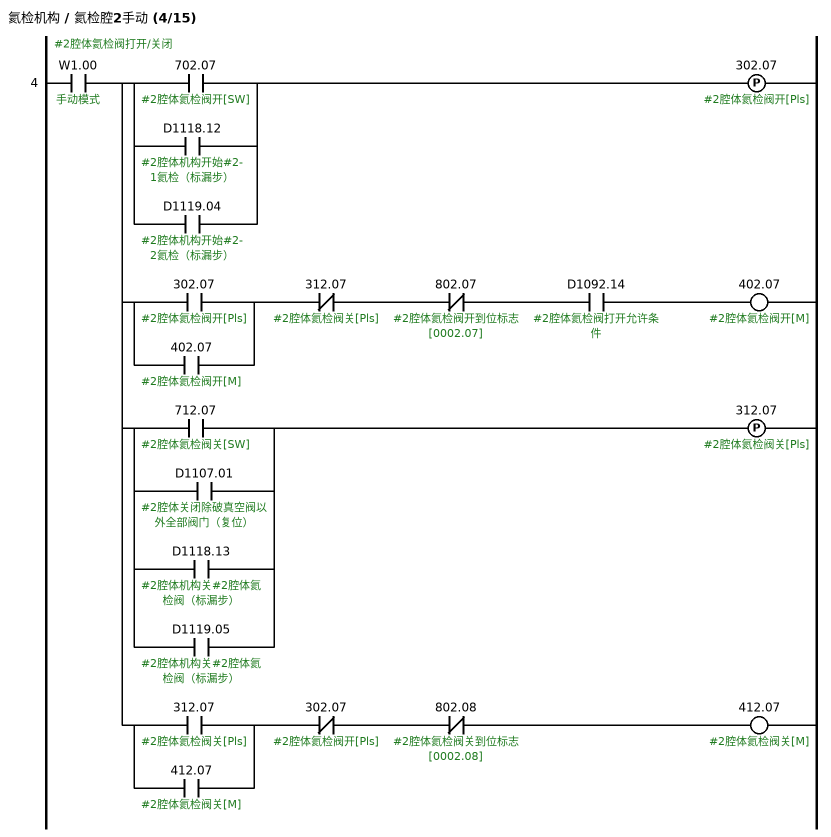
; [picture p168: 氦检机构 / 氦检腔2手动, rungs 4-4]
; rung 4: #2腔体氦检阀打开/关闭
LD W1.00  ; 手动模式
OUT TR0
LD 702.07  ; #2腔体氦检阀开[SW]
OR D1118.12  ; #2腔体机构开始#2-1氦检（标漏步）
OR D1119.04  ; #2腔体机构开始#2-2氦检（标漏步）
ANDLD
DIFU(013) 302.07  ; #2腔体氦检阀开[Pls]
LD TR0
LD 302.07  ; #2腔体氦检阀开[Pls]
OR 402.07  ; #2腔体氦检阀开[M]
ANDLD
ANDNOT 312.07  ; #2腔体氦检阀关[Pls]
ANDNOT 802.07  ; #2腔体氦检阀开到位标志[0002.07]
AND D1092.14  ; #2腔体氦检阀打开允许条件
OUT 402.07  ; #2腔体氦检阀开[M]
LD TR0
LD 712.07  ; #2腔体氦检阀关[SW]
OR D1107.01  ; #2腔体关闭除破真空阀以外全部阀门（复位）
OR D1118.13  ; #2腔体机构关#2腔体氦检阀（标漏步）
OR D1119.05  ; #2腔体机构关#2腔体氦检阀（标漏步）
ANDLD
DIFU(013) 312.07  ; #2腔体氦检阀关[Pls]
LD TR0
LD 312.07  ; #2腔体氦检阀关[Pls]
OR 412.07  ; #2腔体氦检阀关[M]
ANDLD
ANDNOT 302.07  ; #2腔体氦检阀开[Pls]
ANDNOT 802.08  ; #2腔体氦检阀关到位标志[0002.08]
OUT 412.07  ; #2腔体氦检阀关[M]

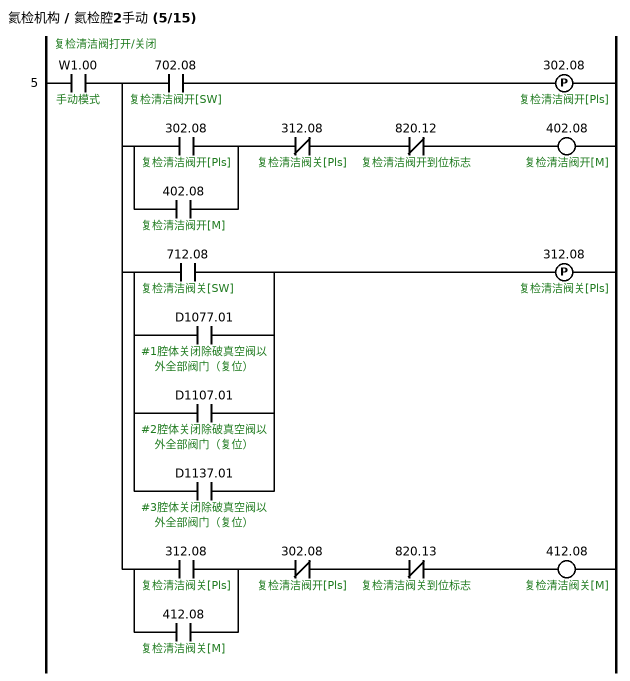
; rung 5: 复检清洁阀打开/关闭
LD W1.00  ; 手动模式
OUT TR0
AND 702.08  ; 复检清洁阀开[SW]
DIFU(013) 302.08  ; 复检清洁阀开[Pls]
LD TR0
LD 302.08  ; 复检清洁阀开[Pls]
OR 402.08  ; 复检清洁阀开[M]
ANDLD
ANDNOT 312.08  ; 复检清洁阀关[Pls]
ANDNOT 820.12  ; 复检清洁阀开到位标志
OUT 402.08  ; 复检清洁阀开[M]
LD TR0
LD 712.08  ; 复检清洁阀关[SW]
OR D1077.01  ; #1腔体关闭除破真空阀以外全部阀门（复位）
OR D1107.01  ; #2腔体关闭除破真空阀以外全部阀门（复位）
OR D1137.01  ; #3腔体关闭除破真空阀以外全部阀门（复位）
ANDLD
DIFU(013) 312.08  ; 复检清洁阀关[Pls]
LD TR0
LD 312.08  ; 复检清洁阀关[Pls]
OR 412.08  ; 复检清洁阀关[M]
ANDLD
ANDNOT 302.08  ; 复检清洁阀开[Pls]
ANDNOT 820.13  ; 复检清洁阀关到位标志
OUT 412.08  ; 复检清洁阀关[M]

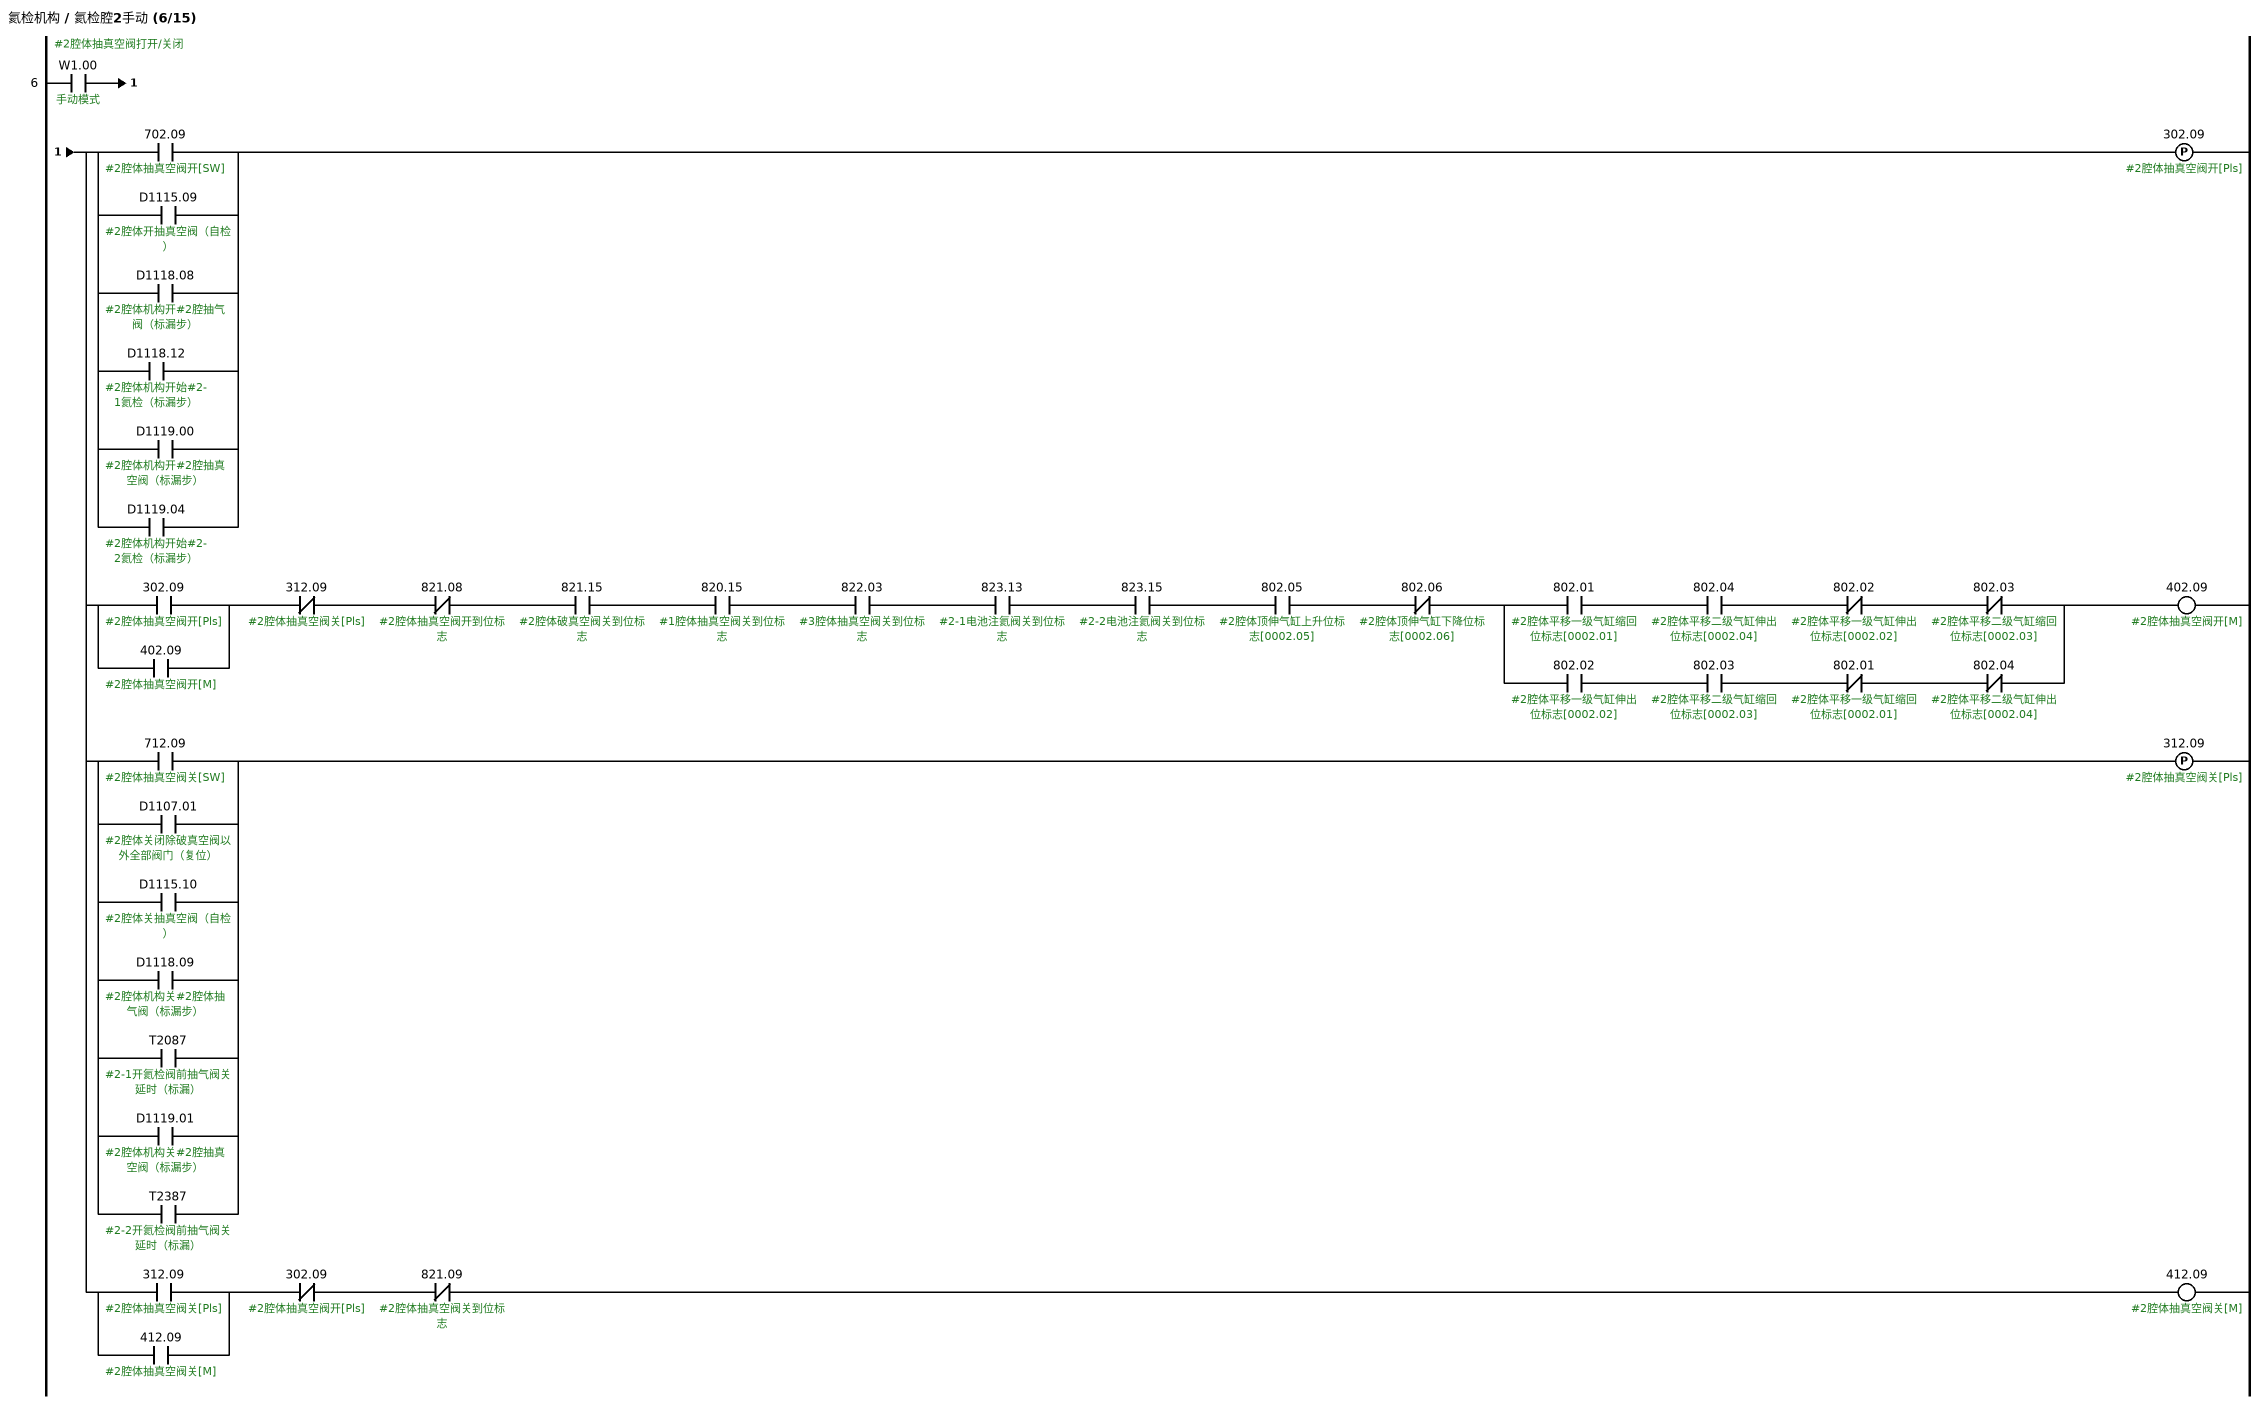
; rung 6: #2腔体抽真空阀打开/关闭
LD W1.00  ; 手动模式
OUT TR0
LD 702.09  ; #2腔体抽真空阀开[SW]
OR D1115.09  ; #2腔体开抽真空阀（自检）
OR D1118.08  ; #2腔体机构开#2腔抽气阀（标漏步）
OR D1118.12  ; #2腔体机构开始#2-1氦检（标漏步）
OR D1119.00  ; #2腔体机构开#2腔抽真空阀（标漏步）
OR D1119.04  ; #2腔体机构开始#2-2氦检（标漏步）
ANDLD
DIFU(013) 302.09  ; #2腔体抽真空阀开[Pls]
LD TR0
LD 302.09  ; #2腔体抽真空阀开[Pls]
OR 402.09  ; #2腔体抽真空阀开[M]
ANDLD
ANDNOT 312.09  ; #2腔体抽真空阀关[Pls]
ANDNOT 821.08  ; #2腔体抽真空阀开到位标志
AND 821.15  ; #2腔体破真空阀关到位标志
AND 820.15  ; #1腔体抽真空阀关到位标志
AND 822.03  ; #3腔体抽真空阀关到位标志
AND 823.13  ; #2-1电池注氦阀关到位标志
AND 823.15  ; #2-2电池注氦阀关到位标志
AND 802.05  ; #2腔体顶伸气缸上升位标志[0002.05]
ANDNOT 802.06  ; #2腔体顶伸气缸下降位标志[0002.06]
LD 802.01  ; #2腔体平移一级气缸缩回位标志[0002.01]
AND 802.04  ; #2腔体平移二级气缸伸出位标志[0002.04]
ANDNOT 802.02  ; #2腔体平移一级气缸伸出位标志[0002.02]
ANDNOT 802.03  ; #2腔体平移二级气缸缩回位标志[0002.03]
LD 802.02  ; #2腔体平移一级气缸伸出位标志[0002.02]
AND 802.03  ; #2腔体平移二级气缸缩回位标志[0002.03]
ANDNOT 802.01  ; #2腔体平移一级气缸缩回位标志[0002.01]
ANDNOT 802.04  ; #2腔体平移二级气缸伸出位标志[0002.04]
ORLD
ANDLD
OUT 402.09  ; #2腔体抽真空阀开[M]
LD TR0
LD 712.09  ; #2腔体抽真空阀关[SW]
OR D1107.01  ; #2腔体关闭除破真空阀以外全部阀门（复位）
OR D1115.10  ; #2腔体关抽真空阀（自检）
OR D1118.09  ; #2腔体机构关#2腔体抽气阀（标漏步）
OR T2087  ; #2-1开氦检阀前抽气阀关延时（标漏）
OR D1119.01  ; #2腔体机构关#2腔抽真空阀（标漏步）
OR T2387  ; #2-2开氦检阀前抽气阀关延时（标漏）
ANDLD
DIFU(013) 312.09  ; #2腔体抽真空阀关[Pls]
LD TR0
LD 312.09  ; #2腔体抽真空阀关[Pls]
OR 412.09  ; #2腔体抽真空阀关[M]
ANDLD
ANDNOT 302.09  ; #2腔体抽真空阀开[Pls]
ANDNOT 821.09  ; #2腔体抽真空阀关到位标志
OUT 412.09  ; #2腔体抽真空阀关[M]

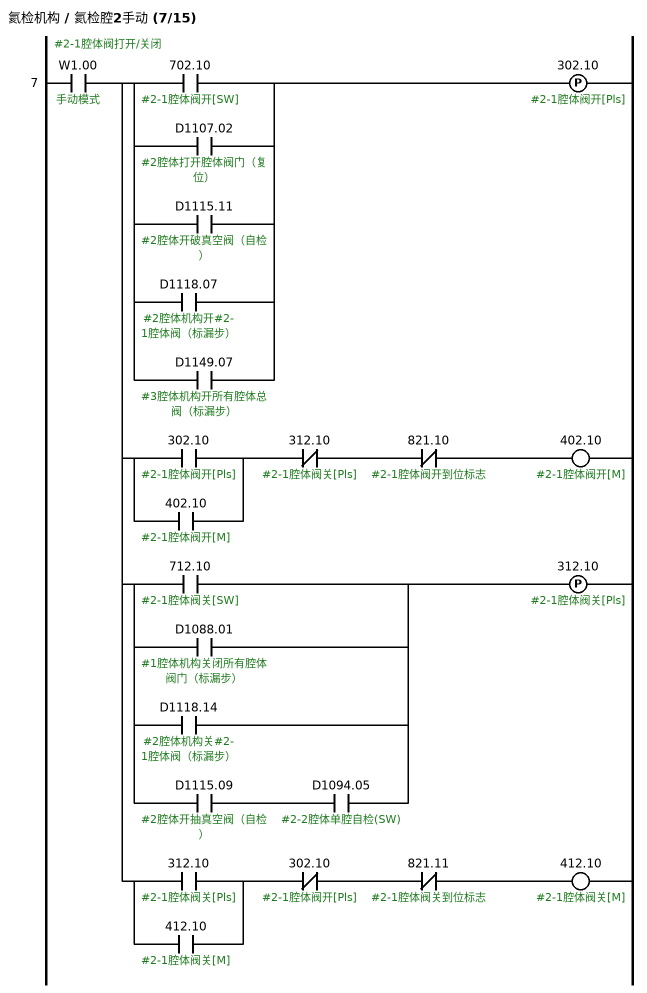
; rung 7: #2-1腔体阀打开/关闭
LD W1.00  ; 手动模式
OUT TR0
LD 702.10  ; #2-1腔体阀开[SW]
OR D1107.02  ; #2腔体打开腔体阀门（复位）
OR D1115.11  ; #2腔体开破真空阀（自检）
OR D1118.07  ; #2腔体机构开#2-1腔体阀（标漏步）
OR D1149.07  ; #3腔体机构开所有腔体总阀（标漏步）
ANDLD
DIFU(013) 302.10  ; #2-1腔体阀开[Pls]
LD TR0
LD 302.10  ; #2-1腔体阀开[Pls]
OR 402.10  ; #2-1腔体阀开[M]
ANDLD
ANDNOT 312.10  ; #2-1腔体阀关[Pls]
ANDNOT 821.10  ; #2-1腔体阀开到位标志
OUT 402.10  ; #2-1腔体阀开[M]
LD TR0
LD 712.10  ; #2-1腔体阀关[SW]
OR D1088.01  ; #1腔体机构关闭所有腔体阀门（标漏步）
OR D1118.14  ; #2腔体机构关#2-1腔体阀（标漏步）
LD D1115.09  ; #2腔体开抽真空阀（自检）
AND D1094.05  ; #2-2腔体单腔自检(SW)
ORLD
ANDLD
DIFU(013) 312.10  ; #2-1腔体阀关[Pls]
LD TR0
LD 312.10  ; #2-1腔体阀关[Pls]
OR 412.10  ; #2-1腔体阀关[M]
ANDLD
ANDNOT 302.10  ; #2-1腔体阀开[Pls]
ANDNOT 821.11  ; #2-1腔体阀关到位标志
OUT 412.10  ; #2-1腔体阀关[M]

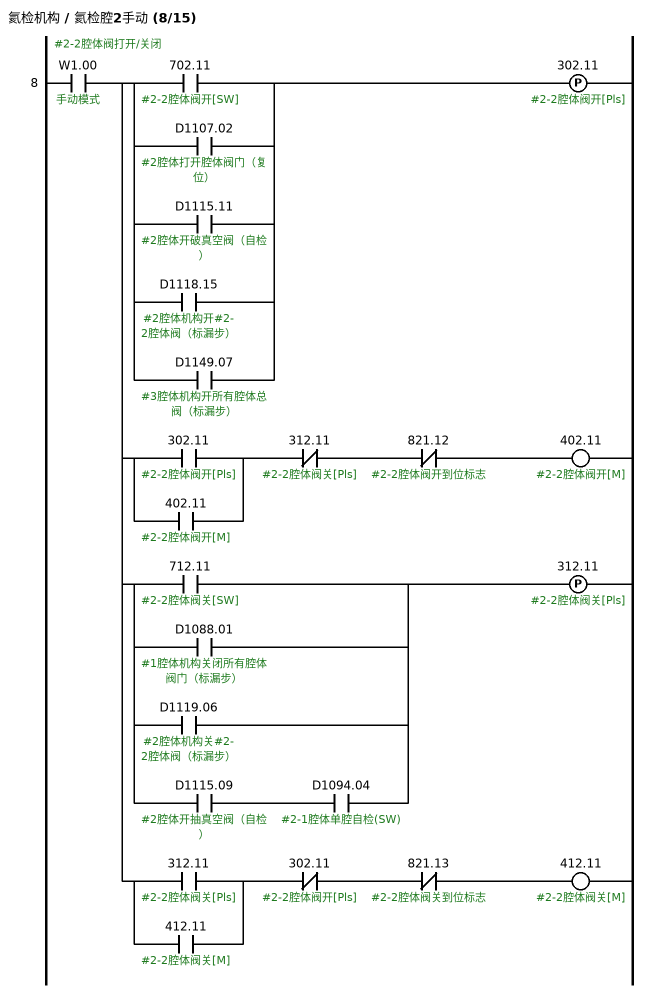
; rung 8: #2-2腔体阀打开/关闭
LD W1.00  ; 手动模式
OUT TR0
LD 702.11  ; #2-2腔体阀开[SW]
OR D1107.02  ; #2腔体打开腔体阀门（复位）
OR D1115.11  ; #2腔体开破真空阀（自检）
OR D1118.15  ; #2腔体机构开#2-2腔体阀（标漏步）
OR D1149.07  ; #3腔体机构开所有腔体总阀（标漏步）
ANDLD
DIFU(013) 302.11  ; #2-2腔体阀开[Pls]
LD TR0
LD 302.11  ; #2-2腔体阀开[Pls]
OR 402.11  ; #2-2腔体阀开[M]
ANDLD
ANDNOT 312.11  ; #2-2腔体阀关[Pls]
ANDNOT 821.12  ; #2-2腔体阀开到位标志
OUT 402.11  ; #2-2腔体阀开[M]
LD TR0
LD 712.11  ; #2-2腔体阀关[SW]
OR D1088.01  ; #1腔体机构关闭所有腔体阀门（标漏步）
OR D1119.06  ; #2腔体机构关#2-2腔体阀（标漏步）
LD D1115.09  ; #2腔体开抽真空阀（自检）
AND D1094.04  ; #2-1腔体单腔自检(SW)
ORLD
ANDLD
DIFU(013) 312.11  ; #2-2腔体阀关[Pls]
LD TR0
LD 312.11  ; #2-2腔体阀关[Pls]
OR 412.11  ; #2-2腔体阀关[M]
ANDLD
ANDNOT 302.11  ; #2-2腔体阀开[Pls]
ANDNOT 821.13  ; #2-2腔体阀关到位标志
OUT 412.11  ; #2-2腔体阀关[M]

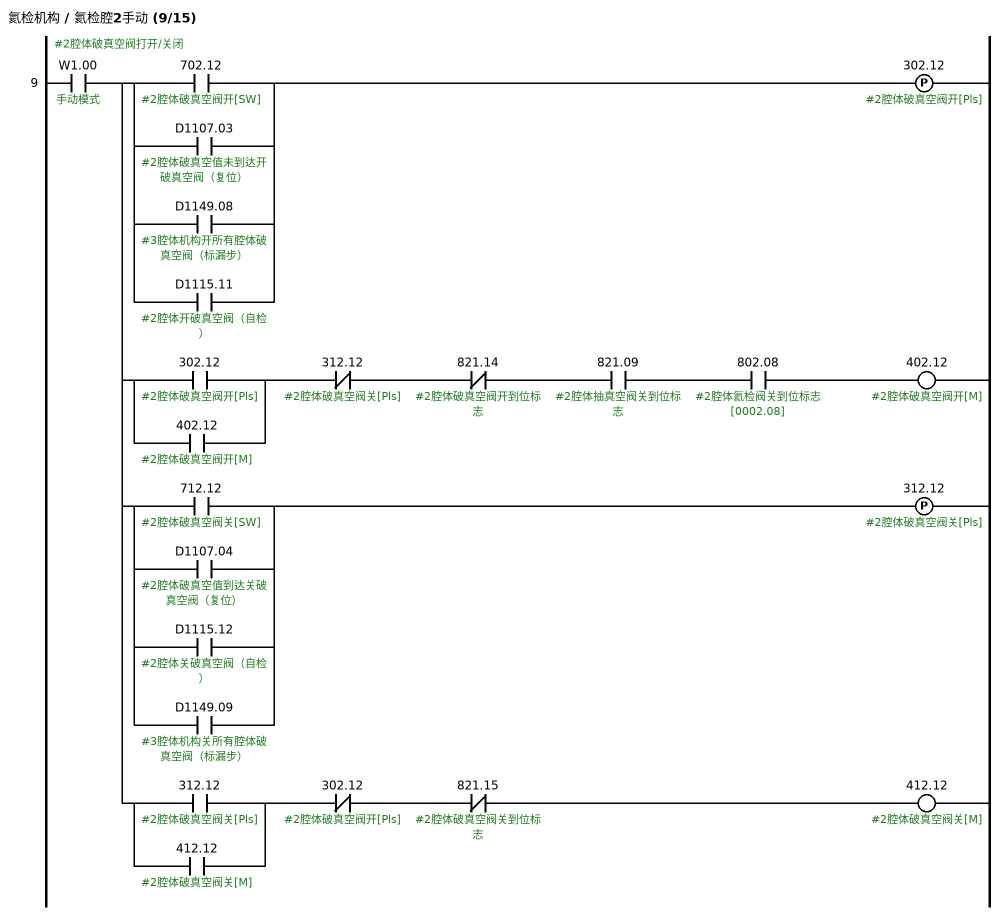
; rung 9: #2腔体破真空阀打开/关闭
LD W1.00  ; 手动模式
OUT TR0
LD 702.12  ; #2腔体破真空阀开[SW]
OR D1107.03  ; #2腔体破真空值未到达开破真空阀（复位）
OR D1149.08  ; #3腔体机构开所有腔体破真空阀（标漏步）
OR D1115.11  ; #2腔体开破真空阀（自检）
ANDLD
DIFU(013) 302.12  ; #2腔体破真空阀开[Pls]
LD TR0
LD 302.12  ; #2腔体破真空阀开[Pls]
OR 402.12  ; #2腔体破真空阀开[M]
ANDLD
ANDNOT 312.12  ; #2腔体破真空阀关[Pls]
ANDNOT 821.14  ; #2腔体破真空阀开到位标志
AND 821.09  ; #2腔体抽真空阀关到位标志
AND 802.08  ; #2腔体氦检阀关到位标志[0002.08]
OUT 402.12  ; #2腔体破真空阀开[M]
LD TR0
LD 712.12  ; #2腔体破真空阀关[SW]
OR D1107.04  ; #2腔体破真空值到达关破真空阀（复位）
OR D1115.12  ; #2腔体关破真空阀（自检）
OR D1149.09  ; #3腔体机构关所有腔体破真空阀（标漏步）
ANDLD
DIFU(013) 312.12  ; #2腔体破真空阀关[Pls]
LD TR0
LD 312.12  ; #2腔体破真空阀关[Pls]
OR 412.12  ; #2腔体破真空阀关[M]
ANDLD
ANDNOT 302.12  ; #2腔体破真空阀开[Pls]
ANDNOT 821.15  ; #2腔体破真空阀关到位标志
OUT 412.12  ; #2腔体破真空阀关[M]

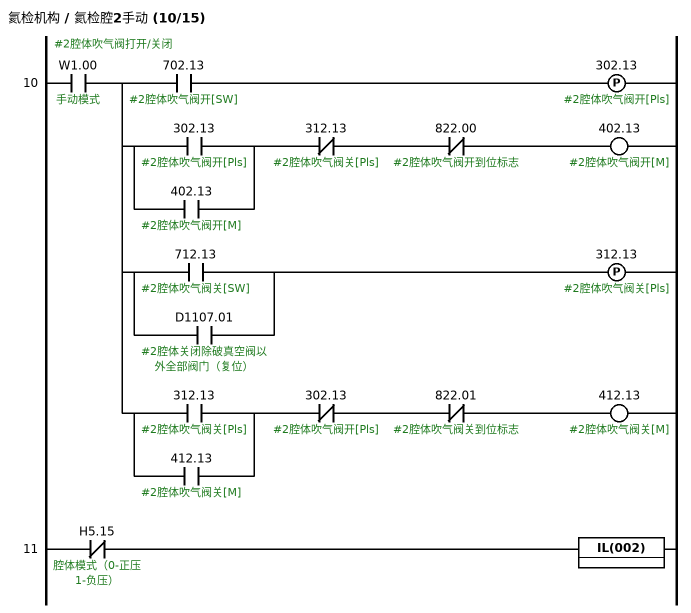
; rung 10: #2腔体吹气阀打开/关闭
LD W1.00  ; 手动模式
OUT TR0
AND 702.13  ; #2腔体吹气阀开[SW]
DIFU(013) 302.13  ; #2腔体吹气阀开[Pls]
LD TR0
LD 302.13  ; #2腔体吹气阀开[Pls]
OR 402.13  ; #2腔体吹气阀开[M]
ANDLD
ANDNOT 312.13  ; #2腔体吹气阀关[Pls]
ANDNOT 822.00  ; #2腔体吹气阀开到位标志
OUT 402.13  ; #2腔体吹气阀开[M]
LD TR0
LD 712.13  ; #2腔体吹气阀关[SW]
OR D1107.01  ; #2腔体关闭除破真空阀以外全部阀门（复位）
ANDLD
DIFU(013) 312.13  ; #2腔体吹气阀关[Pls]
LD TR0
LD 312.13  ; #2腔体吹气阀关[Pls]
OR 412.13  ; #2腔体吹气阀关[M]
ANDLD
ANDNOT 302.13  ; #2腔体吹气阀开[Pls]
ANDNOT 822.01  ; #2腔体吹气阀关到位标志
OUT 412.13  ; #2腔体吹气阀关[M]
; rung 11
LDNOT H5.15  ; 腔体模式（0-正压 1-负压）
IL(002)

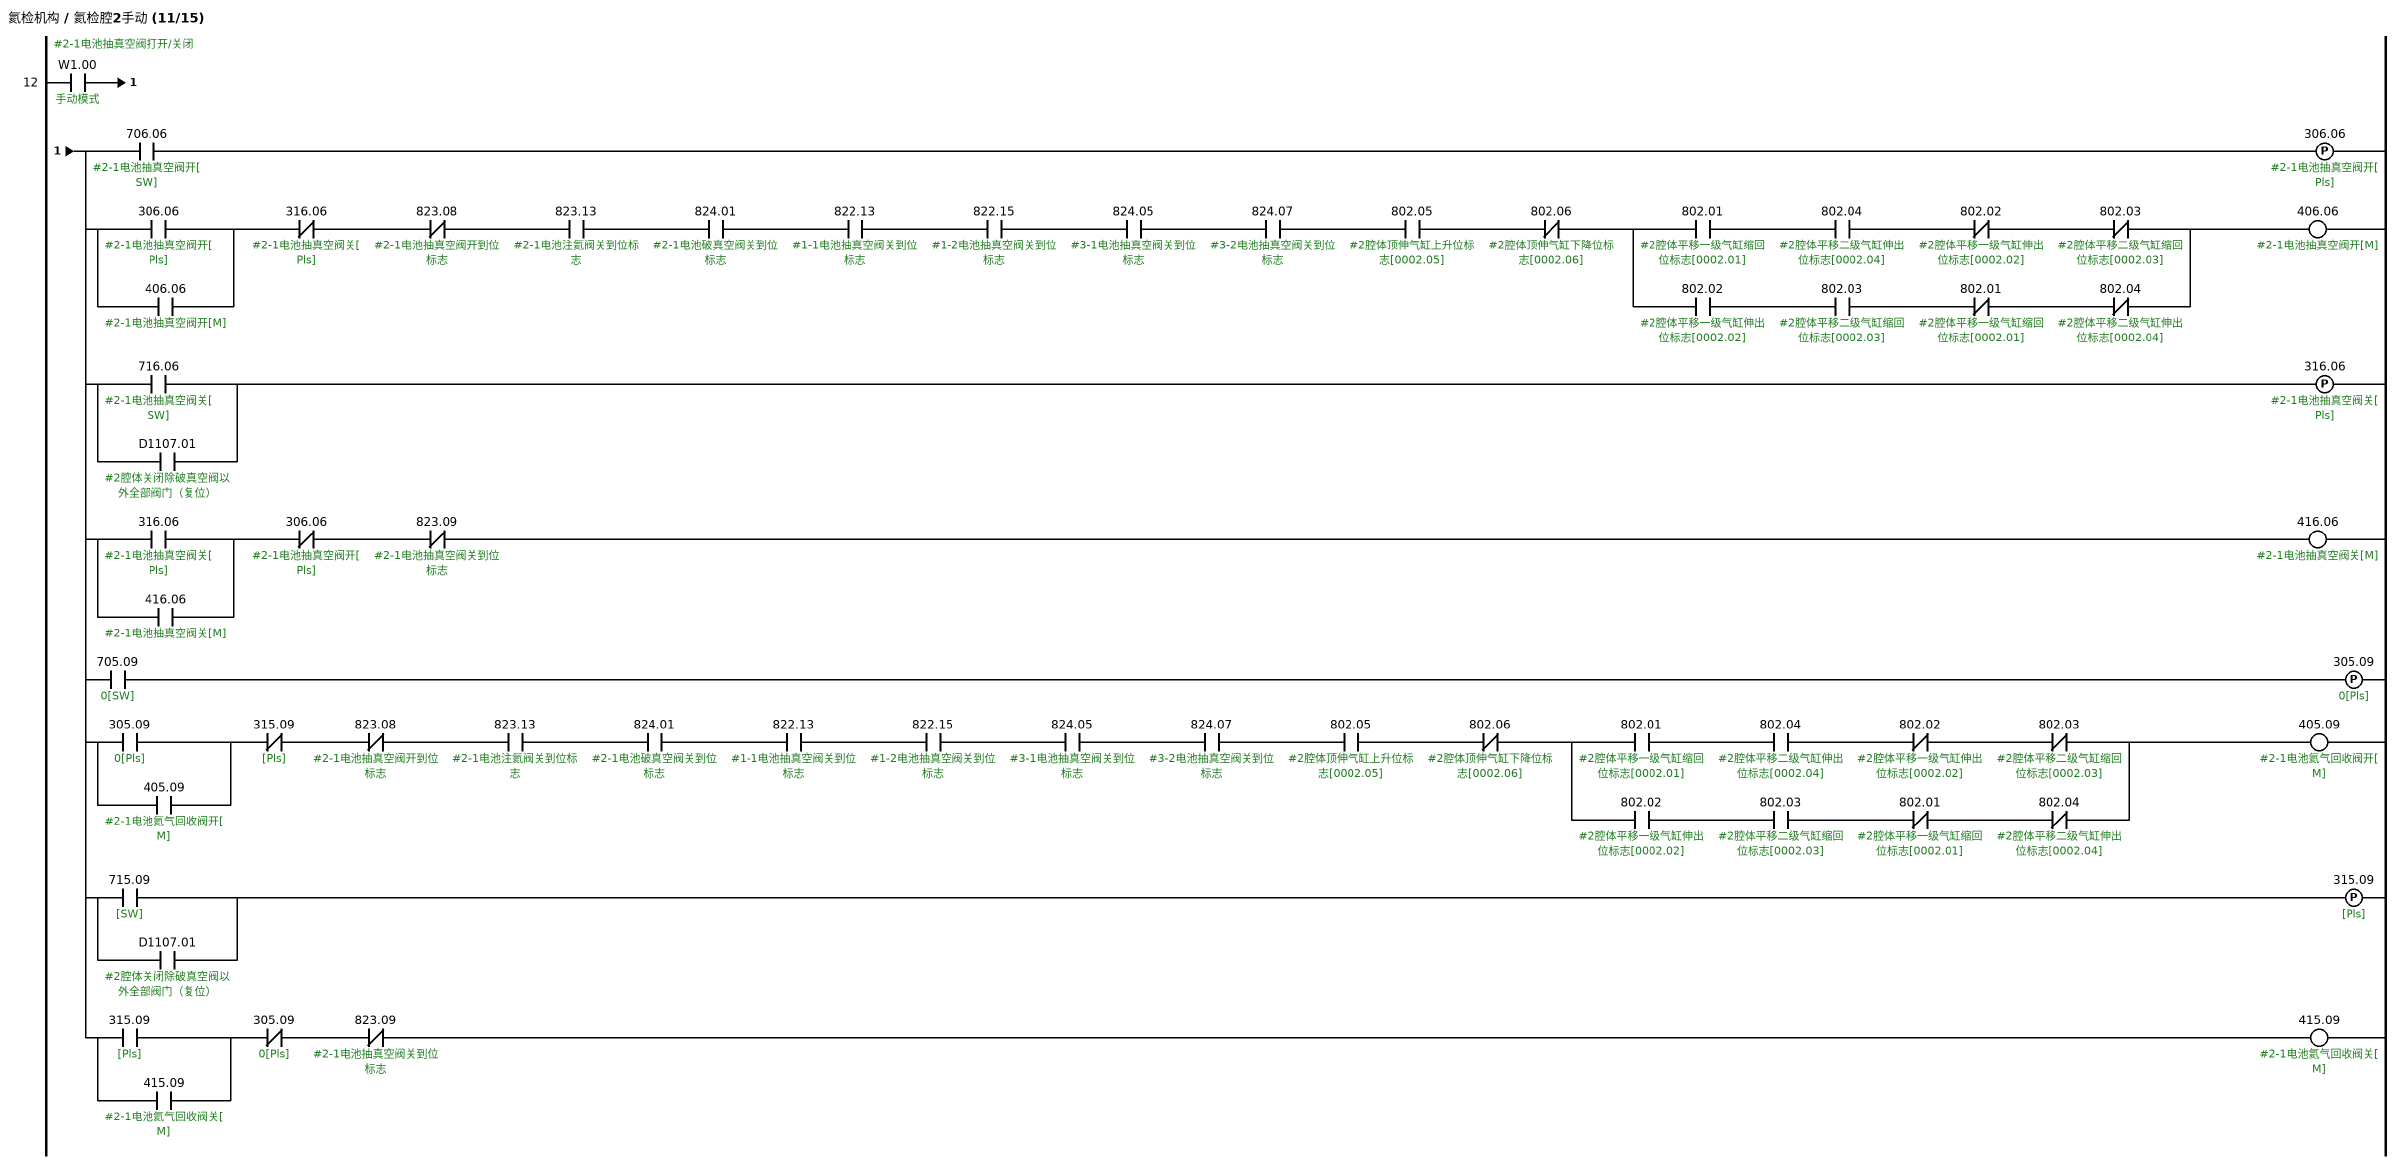
; rung 12: #2-1电池抽真空阀打开/关闭
LD W1.00  ; 手动模式
OUT TR0
AND 706.06  ; #2-1电池抽真空阀开[SW]
DIFU(013) 306.06  ; #2-1电池抽真空阀开[Pls]
LD TR0
LD 306.06  ; #2-1电池抽真空阀开[Pls]
OR 406.06  ; #2-1电池抽真空阀开[M]
ANDLD
ANDNOT 316.06  ; #2-1电池抽真空阀关[Pls]
ANDNOT 823.08  ; #2-1电池抽真空阀开到位标志
AND 823.13  ; #2-1电池注氦阀关到位标志
AND 824.01  ; #2-1电池破真空阀关到位标志
AND 822.13  ; #1-1电池抽真空阀关到位标志
AND 822.15  ; #1-2电池抽真空阀关到位标志
AND 824.05  ; #3-1电池抽真空阀关到位标志
AND 824.07  ; #3-2电池抽真空阀关到位标志
AND 802.05  ; #2腔体顶伸气缸上升位标志[0002.05]
ANDNOT 802.06  ; #2腔体顶伸气缸下降位标志[0002.06]
LD 802.01  ; #2腔体平移一级气缸缩回位标志[0002.01]
AND 802.04  ; #2腔体平移二级气缸伸出位标志[0002.04]
ANDNOT 802.02  ; #2腔体平移一级气缸伸出位标志[0002.02]
ANDNOT 802.03  ; #2腔体平移二级气缸缩回位标志[0002.03]
LD 802.02  ; #2腔体平移一级气缸伸出位标志[0002.02]
AND 802.03  ; #2腔体平移二级气缸缩回位标志[0002.03]
ANDNOT 802.01  ; #2腔体平移一级气缸缩回位标志[0002.01]
ANDNOT 802.04  ; #2腔体平移二级气缸伸出位标志[0002.04]
ORLD
ANDLD
OUT 406.06  ; #2-1电池抽真空阀开[M]
LD TR0
LD 716.06  ; #2-1电池抽真空阀关[SW]
OR D1107.01  ; #2腔体关闭除破真空阀以外全部阀门（复位）
ANDLD
DIFU(013) 316.06  ; #2-1电池抽真空阀关[Pls]
LD TR0
LD 316.06  ; #2-1电池抽真空阀关[Pls]
OR 416.06  ; #2-1电池抽真空阀关[M]
ANDLD
ANDNOT 306.06  ; #2-1电池抽真空阀开[Pls]
ANDNOT 823.09  ; #2-1电池抽真空阀关到位标志
OUT 416.06  ; #2-1电池抽真空阀关[M]
LD TR0
AND 705.09  ; 0[SW]
DIFU(013) 305.09  ; 0[Pls]
LD TR0
LD 305.09  ; 0[Pls]
OR 405.09  ; #2-1电池氦气回收阀开[M]
ANDLD
ANDNOT 315.09  ; [Pls]
ANDNOT 823.08  ; #2-1电池抽真空阀开到位标志
AND 823.13  ; #2-1电池注氦阀关到位标志
AND 824.01  ; #2-1电池破真空阀关到位标志
AND 822.13  ; #1-1电池抽真空阀关到位标志
AND 822.15  ; #1-2电池抽真空阀关到位标志
AND 824.05  ; #3-1电池抽真空阀关到位标志
AND 824.07  ; #3-2电池抽真空阀关到位标志
AND 802.05  ; #2腔体顶伸气缸上升位标志[0002.05]
ANDNOT 802.06  ; #2腔体顶伸气缸下降位标志[0002.06]
LD 802.01  ; #2腔体平移一级气缸缩回位标志[0002.01]
AND 802.04  ; #2腔体平移二级气缸伸出位标志[0002.04]
ANDNOT 802.02  ; #2腔体平移一级气缸伸出位标志[0002.02]
ANDNOT 802.03  ; #2腔体平移二级气缸缩回位标志[0002.03]
LD 802.02  ; #2腔体平移一级气缸伸出位标志[0002.02]
AND 802.03  ; #2腔体平移二级气缸缩回位标志[0002.03]
ANDNOT 802.01  ; #2腔体平移一级气缸缩回位标志[0002.01]
ANDNOT 802.04  ; #2腔体平移二级气缸伸出位标志[0002.04]
ORLD
ANDLD
OUT 405.09  ; #2-1电池氦气回收阀开[M]
LD TR0
LD 715.09  ; [SW]
OR D1107.01  ; #2腔体关闭除破真空阀以外全部阀门（复位）
ANDLD
DIFU(013) 315.09  ; [Pls]
LD TR0
LD 315.09  ; [Pls]
OR 415.09  ; #2-1电池氦气回收阀关[M]
ANDLD
ANDNOT 305.09  ; 0[Pls]
ANDNOT 823.09  ; #2-1电池抽真空阀关到位标志
OUT 415.09  ; #2-1电池氦气回收阀关[M]

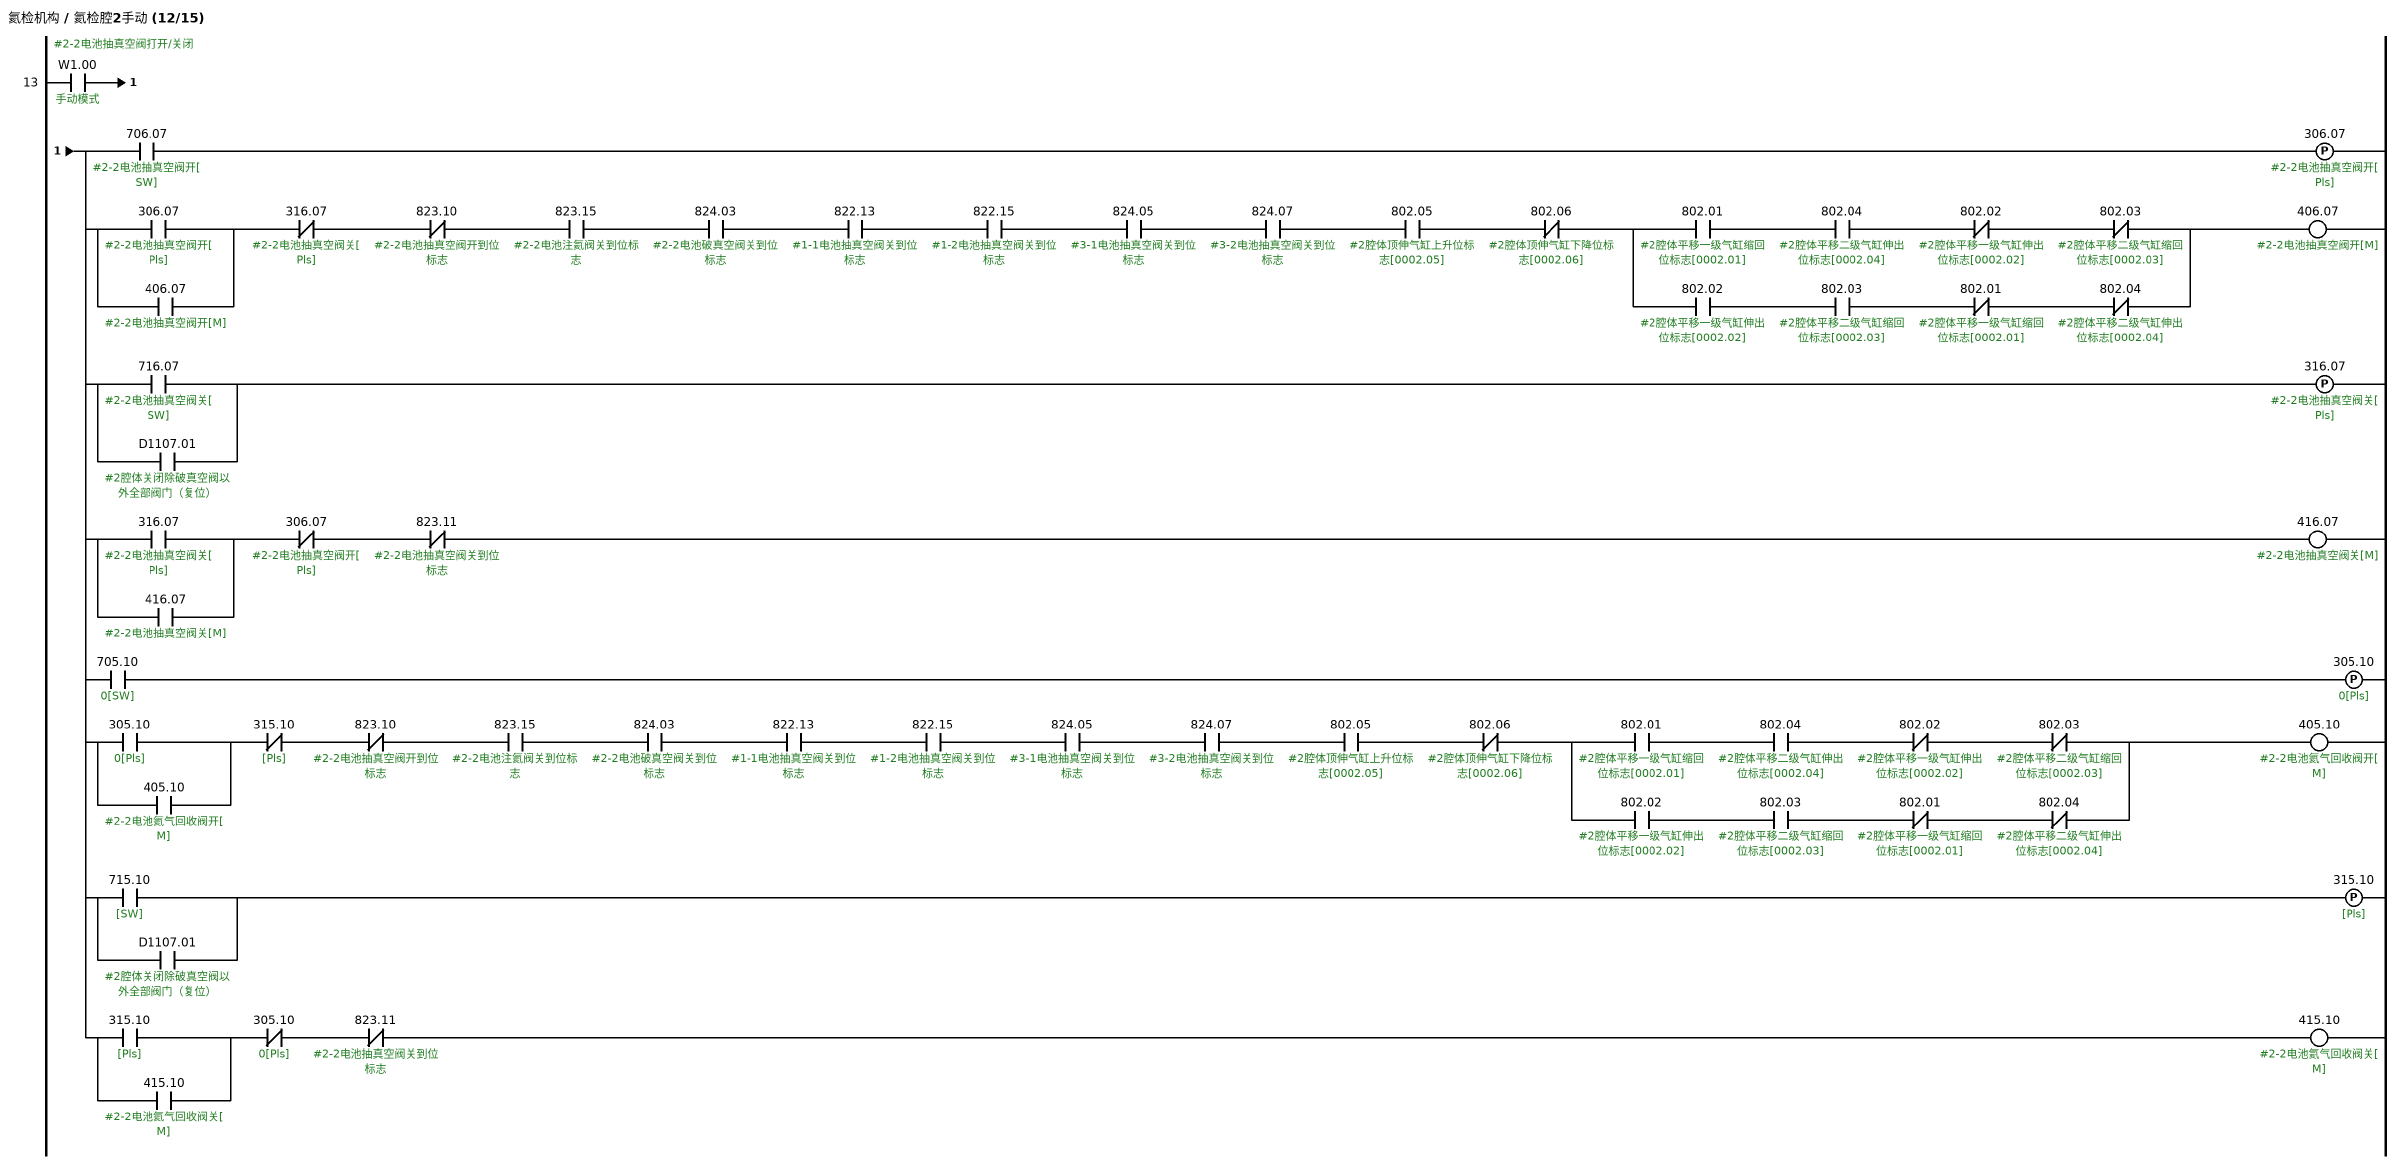
; rung 13: #2-2电池抽真空阀打开/关闭
LD W1.00  ; 手动模式
OUT TR0
AND 706.07  ; #2-2电池抽真空阀开[SW]
DIFU(013) 306.07  ; #2-2电池抽真空阀开[Pls]
LD TR0
LD 306.07  ; #2-2电池抽真空阀开[Pls]
OR 406.07  ; #2-2电池抽真空阀开[M]
ANDLD
ANDNOT 316.07  ; #2-2电池抽真空阀关[Pls]
ANDNOT 823.10  ; #2-2电池抽真空阀开到位标志
AND 823.15  ; #2-2电池注氦阀关到位标志
AND 824.03  ; #2-2电池破真空阀关到位标志
AND 822.13  ; #1-1电池抽真空阀关到位标志
AND 822.15  ; #1-2电池抽真空阀关到位标志
AND 824.05  ; #3-1电池抽真空阀关到位标志
AND 824.07  ; #3-2电池抽真空阀关到位标志
AND 802.05  ; #2腔体顶伸气缸上升位标志[0002.05]
ANDNOT 802.06  ; #2腔体顶伸气缸下降位标志[0002.06]
LD 802.01  ; #2腔体平移一级气缸缩回位标志[0002.01]
AND 802.04  ; #2腔体平移二级气缸伸出位标志[0002.04]
ANDNOT 802.02  ; #2腔体平移一级气缸伸出位标志[0002.02]
ANDNOT 802.03  ; #2腔体平移二级气缸缩回位标志[0002.03]
LD 802.02  ; #2腔体平移一级气缸伸出位标志[0002.02]
AND 802.03  ; #2腔体平移二级气缸缩回位标志[0002.03]
ANDNOT 802.01  ; #2腔体平移一级气缸缩回位标志[0002.01]
ANDNOT 802.04  ; #2腔体平移二级气缸伸出位标志[0002.04]
ORLD
ANDLD
OUT 406.07  ; #2-2电池抽真空阀开[M]
LD TR0
LD 716.07  ; #2-2电池抽真空阀关[SW]
OR D1107.01  ; #2腔体关闭除破真空阀以外全部阀门（复位）
ANDLD
DIFU(013) 316.07  ; #2-2电池抽真空阀关[Pls]
LD TR0
LD 316.07  ; #2-2电池抽真空阀关[Pls]
OR 416.07  ; #2-2电池抽真空阀关[M]
ANDLD
ANDNOT 306.07  ; #2-2电池抽真空阀开[Pls]
ANDNOT 823.11  ; #2-2电池抽真空阀关到位标志
OUT 416.07  ; #2-2电池抽真空阀关[M]
LD TR0
AND 705.10  ; 0[SW]
DIFU(013) 305.10  ; 0[Pls]
LD TR0
LD 305.10  ; 0[Pls]
OR 405.10  ; #2-2电池氦气回收阀开[M]
ANDLD
ANDNOT 315.10  ; [Pls]
ANDNOT 823.10  ; #2-2电池抽真空阀开到位标志
AND 823.15  ; #2-2电池注氦阀关到位标志
AND 824.03  ; #2-2电池破真空阀关到位标志
AND 822.13  ; #1-1电池抽真空阀关到位标志
AND 822.15  ; #1-2电池抽真空阀关到位标志
AND 824.05  ; #3-1电池抽真空阀关到位标志
AND 824.07  ; #3-2电池抽真空阀关到位标志
AND 802.05  ; #2腔体顶伸气缸上升位标志[0002.05]
ANDNOT 802.06  ; #2腔体顶伸气缸下降位标志[0002.06]
LD 802.01  ; #2腔体平移一级气缸缩回位标志[0002.01]
AND 802.04  ; #2腔体平移二级气缸伸出位标志[0002.04]
ANDNOT 802.02  ; #2腔体平移一级气缸伸出位标志[0002.02]
ANDNOT 802.03  ; #2腔体平移二级气缸缩回位标志[0002.03]
LD 802.02  ; #2腔体平移一级气缸伸出位标志[0002.02]
AND 802.03  ; #2腔体平移二级气缸缩回位标志[0002.03]
ANDNOT 802.01  ; #2腔体平移一级气缸缩回位标志[0002.01]
ANDNOT 802.04  ; #2腔体平移二级气缸伸出位标志[0002.04]
ORLD
ANDLD
OUT 405.10  ; #2-2电池氦气回收阀开[M]
LD TR0
LD 715.10  ; [SW]
OR D1107.01  ; #2腔体关闭除破真空阀以外全部阀门（复位）
ANDLD
DIFU(013) 315.10  ; [Pls]
LD TR0
LD 315.10  ; [Pls]
OR 415.10  ; #2-2电池氦气回收阀关[M]
ANDLD
ANDNOT 305.10  ; 0[Pls]
ANDNOT 823.11  ; #2-2电池抽真空阀关到位标志
OUT 415.10  ; #2-2电池氦气回收阀关[M]

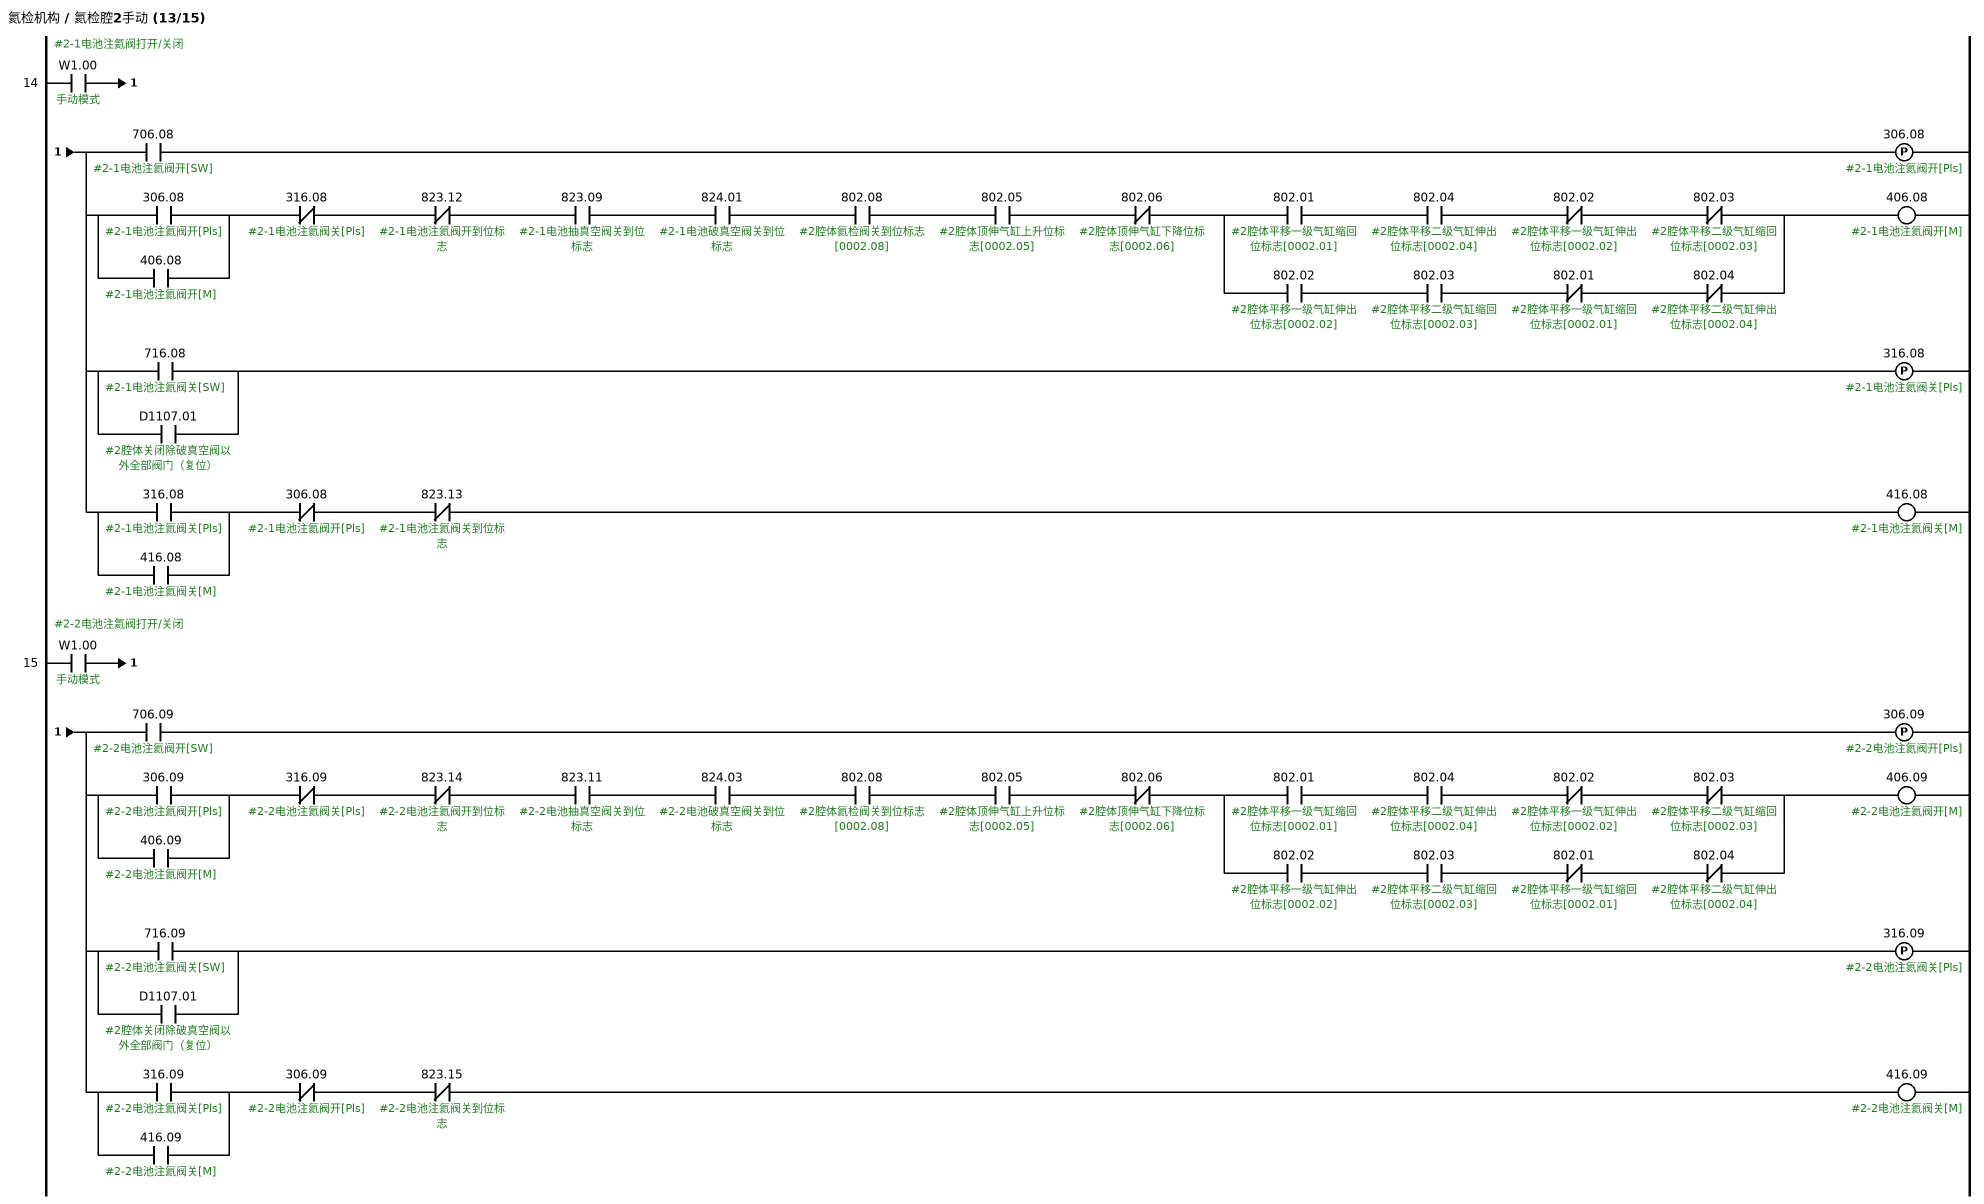
; rung 14: #2-1电池注氦阀打开/关闭
LD W1.00  ; 手动模式
OUT TR0
AND 706.08  ; #2-1电池注氦阀开[SW]
DIFU(013) 306.08  ; #2-1电池注氦阀开[Pls]
LD TR0
LD 306.08  ; #2-1电池注氦阀开[Pls]
OR 406.08  ; #2-1电池注氦阀开[M]
ANDLD
ANDNOT 316.08  ; #2-1电池注氦阀关[Pls]
ANDNOT 823.12  ; #2-1电池注氦阀开到位标志
AND 823.09  ; #2-1电池抽真空阀关到位标志
AND 824.01  ; #2-1电池破真空阀关到位标志
AND 802.08  ; #2腔体氦检阀关到位标志[0002.08]
AND 802.05  ; #2腔体顶伸气缸上升位标志[0002.05]
ANDNOT 802.06  ; #2腔体顶伸气缸下降位标志[0002.06]
LD 802.01  ; #2腔体平移一级气缸缩回位标志[0002.01]
AND 802.04  ; #2腔体平移二级气缸伸出位标志[0002.04]
ANDNOT 802.02  ; #2腔体平移一级气缸伸出位标志[0002.02]
ANDNOT 802.03  ; #2腔体平移二级气缸缩回位标志[0002.03]
LD 802.02  ; #2腔体平移一级气缸伸出位标志[0002.02]
AND 802.03  ; #2腔体平移二级气缸缩回位标志[0002.03]
ANDNOT 802.01  ; #2腔体平移一级气缸缩回位标志[0002.01]
ANDNOT 802.04  ; #2腔体平移二级气缸伸出位标志[0002.04]
ORLD
ANDLD
OUT 406.08  ; #2-1电池注氦阀开[M]
LD TR0
LD 716.08  ; #2-1电池注氦阀关[SW]
OR D1107.01  ; #2腔体关闭除破真空阀以外全部阀门（复位）
ANDLD
DIFU(013) 316.08  ; #2-1电池注氦阀关[Pls]
LD TR0
LD 316.08  ; #2-1电池注氦阀关[Pls]
OR 416.08  ; #2-1电池注氦阀关[M]
ANDLD
ANDNOT 306.08  ; #2-1电池注氦阀开[Pls]
ANDNOT 823.13  ; #2-1电池注氦阀关到位标志
OUT 416.08  ; #2-1电池注氦阀关[M]
; rung 15: #2-2电池注氦阀打开/关闭
LD W1.00  ; 手动模式
OUT TR0
AND 706.09  ; #2-2电池注氦阀开[SW]
DIFU(013) 306.09  ; #2-2电池注氦阀开[Pls]
LD TR0
LD 306.09  ; #2-2电池注氦阀开[Pls]
OR 406.09  ; #2-2电池注氦阀开[M]
ANDLD
ANDNOT 316.09  ; #2-2电池注氦阀关[Pls]
ANDNOT 823.14  ; #2-2电池注氦阀开到位标志
AND 823.11  ; #2-2电池抽真空阀关到位标志
AND 824.03  ; #2-2电池破真空阀关到位标志
AND 802.08  ; #2腔体氦检阀关到位标志[0002.08]
AND 802.05  ; #2腔体顶伸气缸上升位标志[0002.05]
ANDNOT 802.06  ; #2腔体顶伸气缸下降位标志[0002.06]
LD 802.01  ; #2腔体平移一级气缸缩回位标志[0002.01]
AND 802.04  ; #2腔体平移二级气缸伸出位标志[0002.04]
ANDNOT 802.02  ; #2腔体平移一级气缸伸出位标志[0002.02]
ANDNOT 802.03  ; #2腔体平移二级气缸缩回位标志[0002.03]
LD 802.02  ; #2腔体平移一级气缸伸出位标志[0002.02]
AND 802.03  ; #2腔体平移二级气缸缩回位标志[0002.03]
ANDNOT 802.01  ; #2腔体平移一级气缸缩回位标志[0002.01]
ANDNOT 802.04  ; #2腔体平移二级气缸伸出位标志[0002.04]
ORLD
ANDLD
OUT 406.09  ; #2-2电池注氦阀开[M]
LD TR0
LD 716.09  ; #2-2电池注氦阀关[SW]
OR D1107.01  ; #2腔体关闭除破真空阀以外全部阀门（复位）
ANDLD
DIFU(013) 316.09  ; #2-2电池注氦阀关[Pls]
LD TR0
LD 316.09  ; #2-2电池注氦阀关[Pls]
OR 416.09  ; #2-2电池注氦阀关[M]
ANDLD
ANDNOT 306.09  ; #2-2电池注氦阀开[Pls]
ANDNOT 823.15  ; #2-2电池注氦阀关到位标志
OUT 416.09  ; #2-2电池注氦阀关[M]

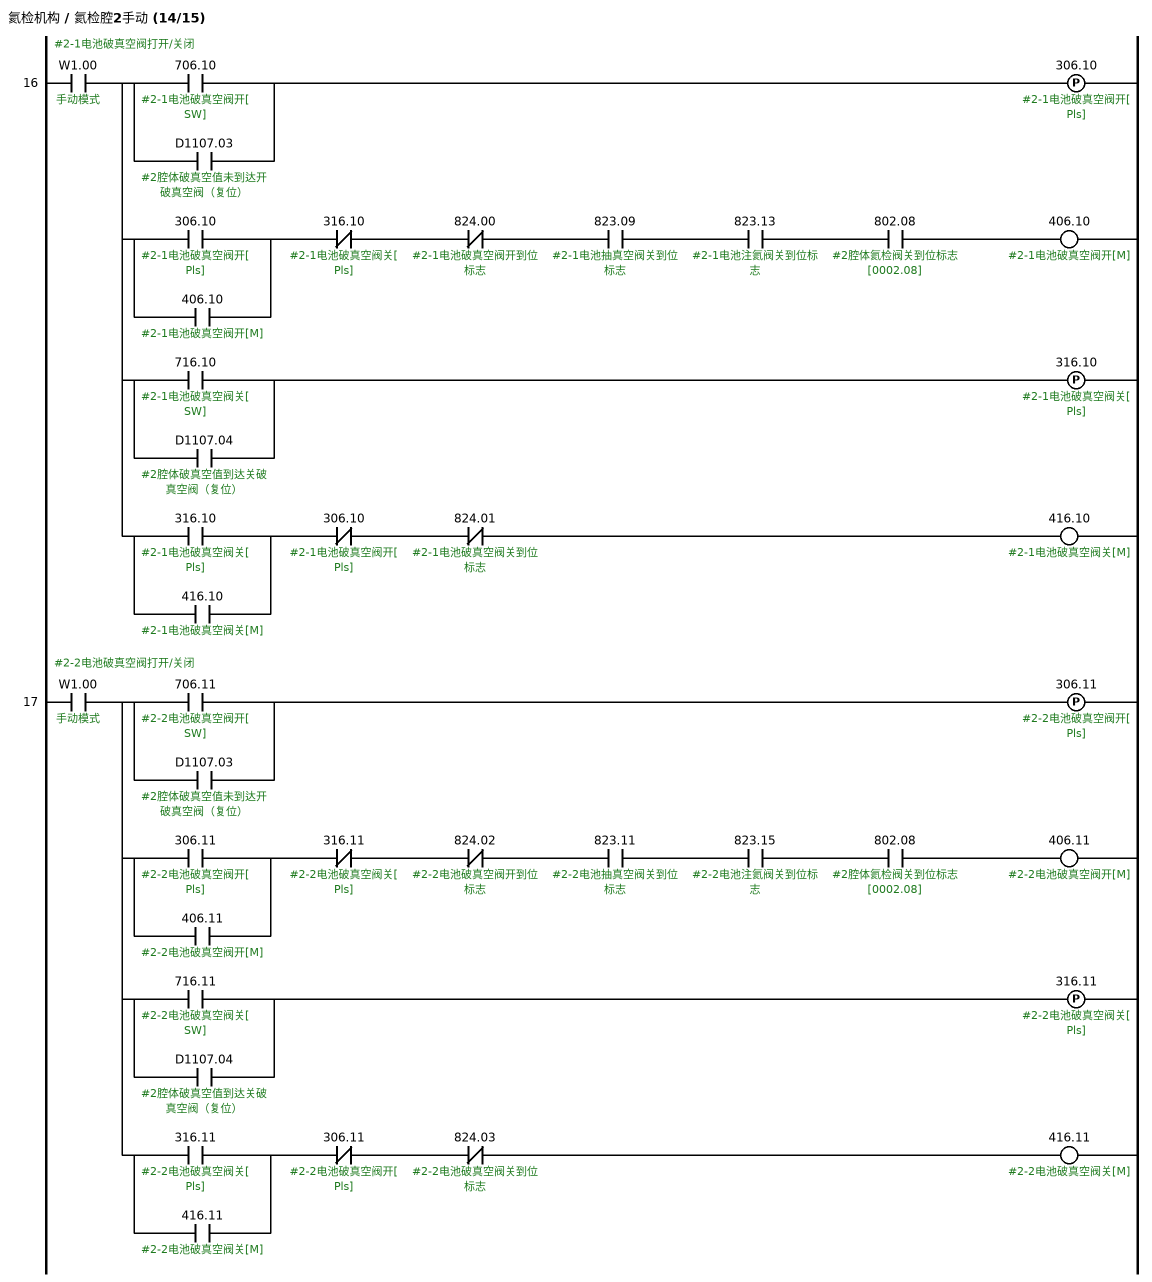
; rung 16: #2-1电池破真空阀打开/关闭
LD W1.00  ; 手动模式
OUT TR0
LD 706.10  ; #2-1电池破真空阀开[SW]
OR D1107.03  ; #2腔体破真空值未到达开破真空阀（复位）
ANDLD
DIFU(013) 306.10  ; #2-1电池破真空阀开[Pls]
LD TR0
LD 306.10  ; #2-1电池破真空阀开[Pls]
OR 406.10  ; #2-1电池破真空阀开[M]
ANDLD
ANDNOT 316.10  ; #2-1电池破真空阀关[Pls]
ANDNOT 824.00  ; #2-1电池破真空阀开到位标志
AND 823.09  ; #2-1电池抽真空阀关到位标志
AND 823.13  ; #2-1电池注氦阀关到位标志
AND 802.08  ; #2腔体氦检阀关到位标志[0002.08]
OUT 406.10  ; #2-1电池破真空阀开[M]
LD TR0
LD 716.10  ; #2-1电池破真空阀关[SW]
OR D1107.04  ; #2腔体破真空值到达关破真空阀（复位）
ANDLD
DIFU(013) 316.10  ; #2-1电池破真空阀关[Pls]
LD TR0
LD 316.10  ; #2-1电池破真空阀关[Pls]
OR 416.10  ; #2-1电池破真空阀关[M]
ANDLD
ANDNOT 306.10  ; #2-1电池破真空阀开[Pls]
ANDNOT 824.01  ; #2-1电池破真空阀关到位标志
OUT 416.10  ; #2-1电池破真空阀关[M]
; rung 17: #2-2电池破真空阀打开/关闭
LD W1.00  ; 手动模式
OUT TR0
LD 706.11  ; #2-2电池破真空阀开[SW]
OR D1107.03  ; #2腔体破真空值未到达开破真空阀（复位）
ANDLD
DIFU(013) 306.11  ; #2-2电池破真空阀开[Pls]
LD TR0
LD 306.11  ; #2-2电池破真空阀开[Pls]
OR 406.11  ; #2-2电池破真空阀开[M]
ANDLD
ANDNOT 316.11  ; #2-2电池破真空阀关[Pls]
ANDNOT 824.02  ; #2-2电池破真空阀开到位标志
AND 823.11  ; #2-2电池抽真空阀关到位标志
AND 823.15  ; #2-2电池注氦阀关到位标志
AND 802.08  ; #2腔体氦检阀关到位标志[0002.08]
OUT 406.11  ; #2-2电池破真空阀开[M]
LD TR0
LD 716.11  ; #2-2电池破真空阀关[SW]
OR D1107.04  ; #2腔体破真空值到达关破真空阀（复位）
ANDLD
DIFU(013) 316.11  ; #2-2电池破真空阀关[Pls]
LD TR0
LD 316.11  ; #2-2电池破真空阀关[Pls]
OR 416.11  ; #2-2电池破真空阀关[M]
ANDLD
ANDNOT 306.11  ; #2-2电池破真空阀开[Pls]
ANDNOT 824.03  ; #2-2电池破真空阀关到位标志
OUT 416.11  ; #2-2电池破真空阀关[M]

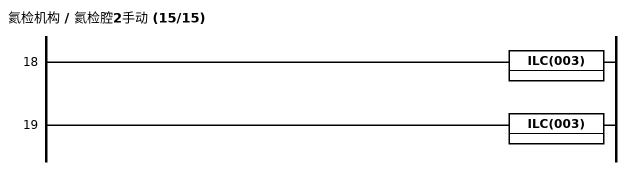
; rung 18
ILC(003)
; rung 19
ILC(003)

### Section 氦检腔3手动

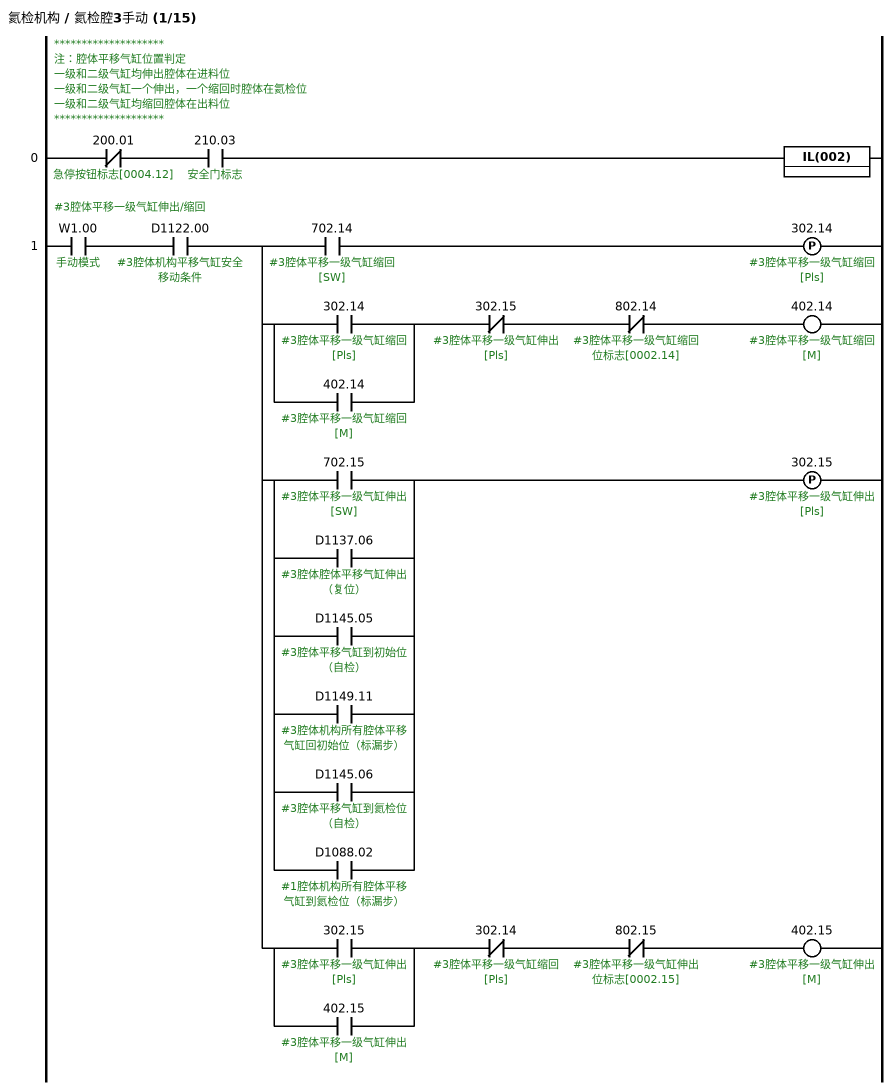
; rung 0: ******************** / 注：腔体平移气缸位置判定 / 一级和二级气缸均伸出腔体在进料位 / 一级和二级气缸一个伸出，一个缩回时腔体在氦检位 / 一级和二级气缸均缩回腔体在出料位 / ********************
LDNOT 200.01  ; 急停按钮标志[0004.12]
AND 210.03  ; 安全门标志
IL(002)
; rung 1: #3腔体平移一级气缸伸出/缩回
LD W1.00  ; 手动模式
AND D1122.00  ; #3腔体机构平移气缸安全移动条件
OUT TR0
AND 702.14  ; #3腔体平移一级气缸缩回[SW]
DIFU(013) 302.14  ; #3腔体平移一级气缸缩回[Pls]
LD TR0
LD 302.14  ; #3腔体平移一级气缸缩回[Pls]
OR 402.14  ; #3腔体平移一级气缸缩回[M]
ANDLD
ANDNOT 302.15  ; #3腔体平移一级气缸伸出[Pls]
ANDNOT 802.14  ; #3腔体平移一级气缸缩回位标志[0002.14]
OUT 402.14  ; #3腔体平移一级气缸缩回[M]
LD TR0
LD 702.15  ; #3腔体平移一级气缸伸出[SW]
OR D1137.06  ; #3腔体腔体平移气缸伸出（复位）
OR D1145.05  ; #3腔体平移气缸到初始位（自检）
OR D1149.11  ; #3腔体机构所有腔体平移气缸回初始位（标漏步）
OR D1145.06  ; #3腔体平移气缸到氦检位（自检）
OR D1088.02  ; #1腔体机构所有腔体平移气缸到氦检位（标漏步）
ANDLD
DIFU(013) 302.15  ; #3腔体平移一级气缸伸出[Pls]
LD TR0
LD 302.15  ; #3腔体平移一级气缸伸出[Pls]
OR 402.15  ; #3腔体平移一级气缸伸出[M]
ANDLD
ANDNOT 302.14  ; #3腔体平移一级气缸缩回[Pls]
ANDNOT 802.15  ; #3腔体平移一级气缸伸出位标志[0002.15]
OUT 402.15  ; #3腔体平移一级气缸伸出[M]

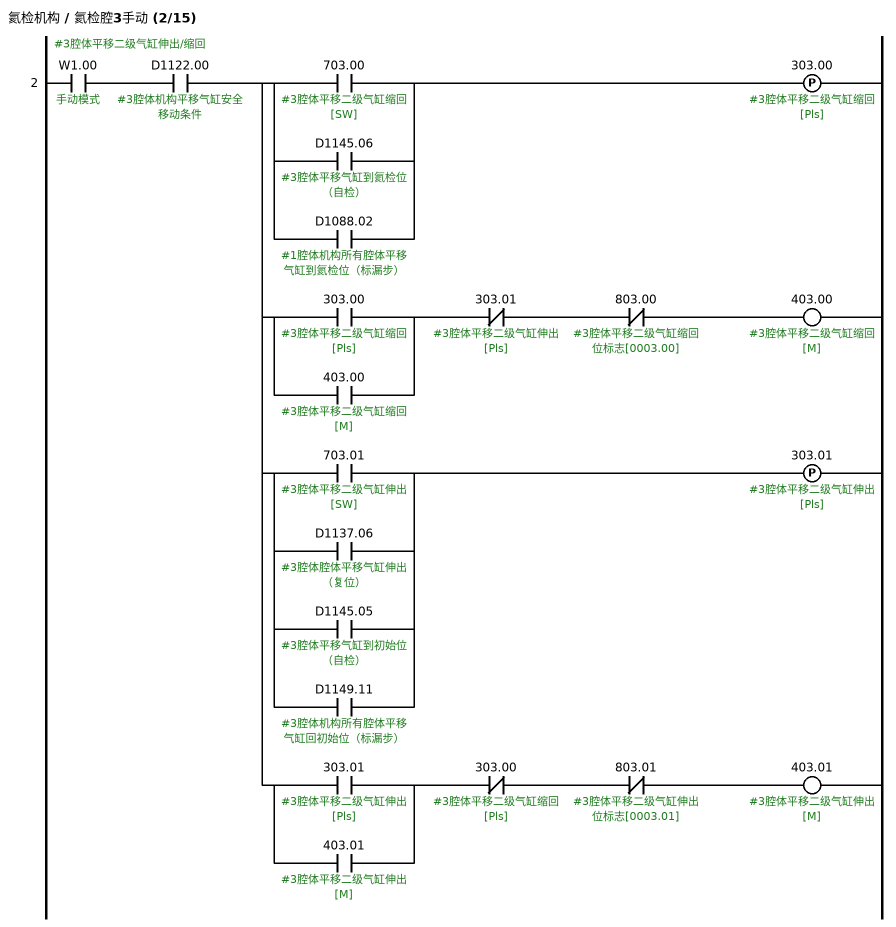
; rung 2: #3腔体平移二级气缸伸出/缩回
LD W1.00  ; 手动模式
AND D1122.00  ; #3腔体机构平移气缸安全移动条件
OUT TR0
LD 703.00  ; #3腔体平移二级气缸缩回[SW]
OR D1145.06  ; #3腔体平移气缸到氦检位（自检）
OR D1088.02  ; #1腔体机构所有腔体平移气缸到氦检位（标漏步）
ANDLD
DIFU(013) 303.00  ; #3腔体平移二级气缸缩回[Pls]
LD TR0
LD 303.00  ; #3腔体平移二级气缸缩回[Pls]
OR 403.00  ; #3腔体平移二级气缸缩回[M]
ANDLD
ANDNOT 303.01  ; #3腔体平移二级气缸伸出[Pls]
ANDNOT 803.00  ; #3腔体平移二级气缸缩回位标志[0003.00]
OUT 403.00  ; #3腔体平移二级气缸缩回[M]
LD TR0
LD 703.01  ; #3腔体平移二级气缸伸出[SW]
OR D1137.06  ; #3腔体腔体平移气缸伸出（复位）
OR D1145.05  ; #3腔体平移气缸到初始位（自检）
OR D1149.11  ; #3腔体机构所有腔体平移气缸回初始位（标漏步）
ANDLD
DIFU(013) 303.01  ; #3腔体平移二级气缸伸出[Pls]
LD TR0
LD 303.01  ; #3腔体平移二级气缸伸出[Pls]
OR 403.01  ; #3腔体平移二级气缸伸出[M]
ANDLD
ANDNOT 303.00  ; #3腔体平移二级气缸缩回[Pls]
ANDNOT 803.01  ; #3腔体平移二级气缸伸出位标志[0003.01]
OUT 403.01  ; #3腔体平移二级气缸伸出[M]

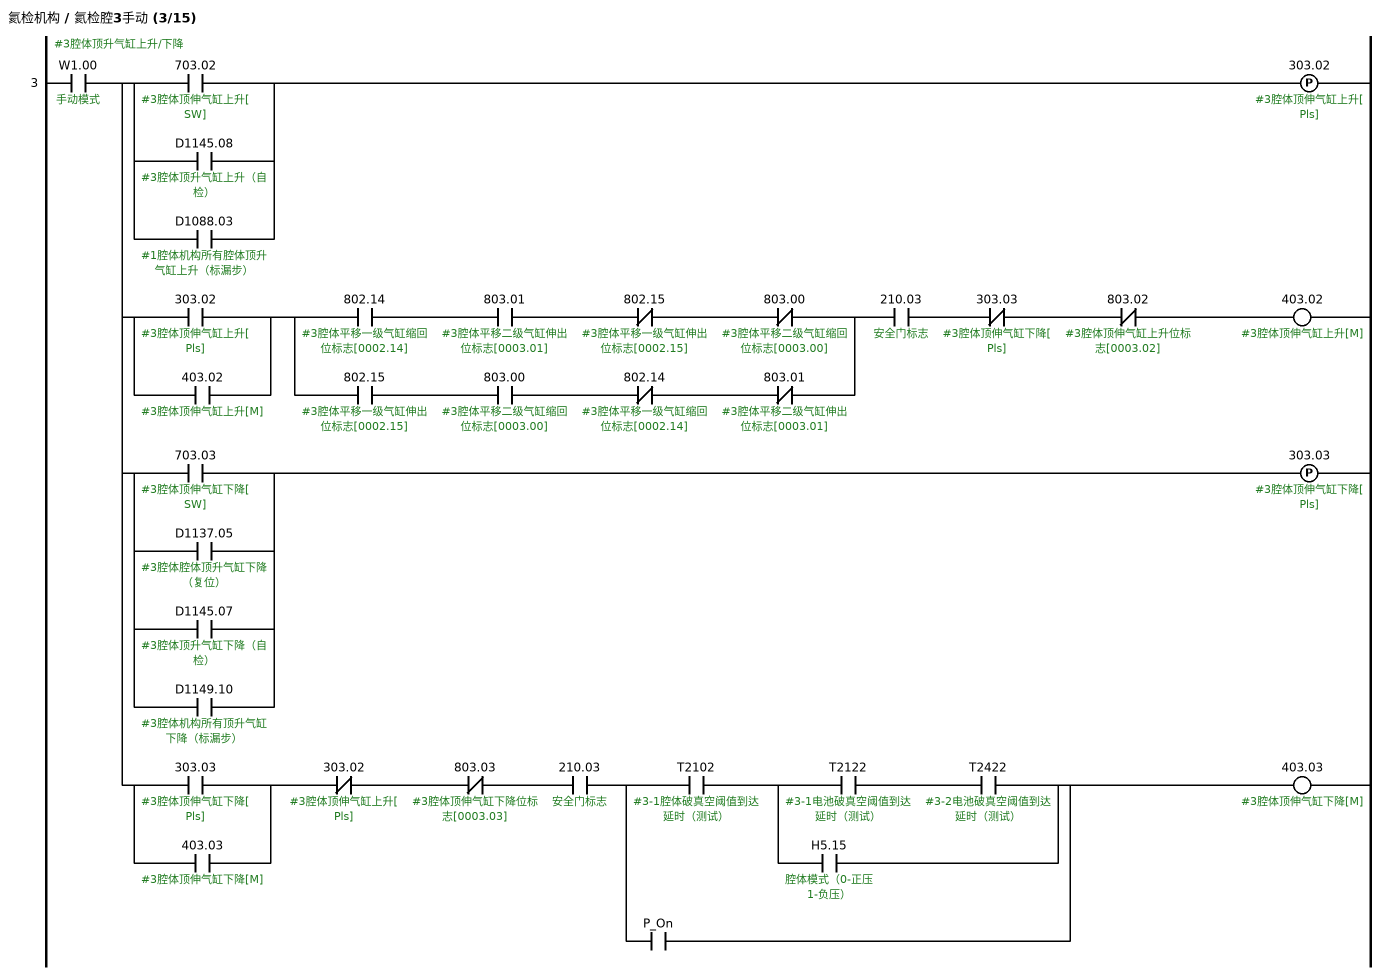
; rung 3: #3腔体顶升气缸上升/下降
LD W1.00  ; 手动模式
OUT TR0
LD 703.02  ; #3腔体顶伸气缸上升[SW]
OR D1145.08  ; #3腔体顶升气缸上升（自检）
OR D1088.03  ; #1腔体机构所有腔体顶升气缸上升（标漏步）
ANDLD
DIFU(013) 303.02  ; #3腔体顶伸气缸上升[Pls]
LD TR0
LD 303.02  ; #3腔体顶伸气缸上升[Pls]
OR 403.02  ; #3腔体顶伸气缸上升[M]
ANDLD
LD 802.14  ; #3腔体平移一级气缸缩回位标志[0002.14]
AND 803.01  ; #3腔体平移二级气缸伸出位标志[0003.01]
ANDNOT 802.15  ; #3腔体平移一级气缸伸出位标志[0002.15]
ANDNOT 803.00  ; #3腔体平移二级气缸缩回位标志[0003.00]
LD 802.15  ; #3腔体平移一级气缸伸出位标志[0002.15]
AND 803.00  ; #3腔体平移二级气缸缩回位标志[0003.00]
ANDNOT 802.14  ; #3腔体平移一级气缸缩回位标志[0002.14]
ANDNOT 803.01  ; #3腔体平移二级气缸伸出位标志[0003.01]
ORLD
ANDLD
AND 210.03  ; 安全门标志
ANDNOT 303.03  ; #3腔体顶伸气缸下降[Pls]
ANDNOT 803.02  ; #3腔体顶伸气缸上升位标志[0003.02]
OUT 403.02  ; #3腔体顶伸气缸上升[M]
LD TR0
LD 703.03  ; #3腔体顶伸气缸下降[SW]
OR D1137.05  ; #3腔体腔体顶升气缸下降（复位）
OR D1145.07  ; #3腔体顶升气缸下降（自检）
OR D1149.10  ; #3腔体机构所有顶升气缸下降（标漏步）
ANDLD
DIFU(013) 303.03  ; #3腔体顶伸气缸下降[Pls]
LD TR0
LD 303.03  ; #3腔体顶伸气缸下降[Pls]
OR 403.03  ; #3腔体顶伸气缸下降[M]
ANDLD
ANDNOT 303.02  ; #3腔体顶伸气缸上升[Pls]
ANDNOT 803.03  ; #3腔体顶伸气缸下降位标志[0003.03]
AND 210.03  ; 安全门标志
LD T2102  ; #3-1腔体破真空阈值到达延时（测试）
LD T2122  ; #3-1电池破真空阈值到达延时（测试）
AND T2422  ; #3-2电池破真空阈值到达延时（测试）
OR H5.15  ; 腔体模式（0-正压 1-负压）
ANDLD
OR P_On
ANDLD
OUT 403.03  ; #3腔体顶伸气缸下降[M]

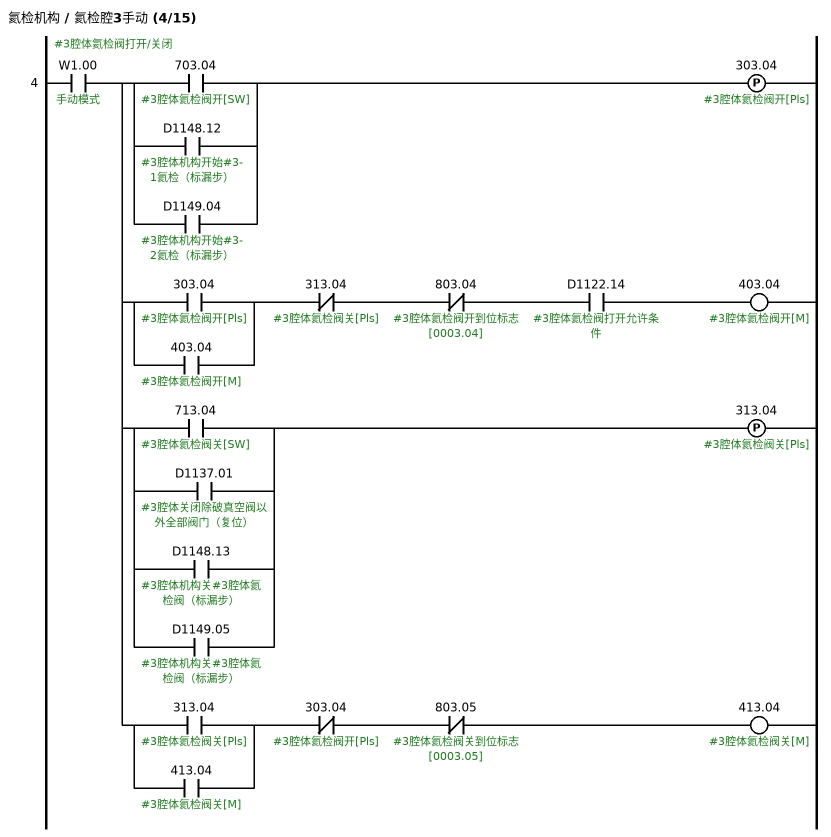
; rung 4: #3腔体氦检阀打开/关闭
LD W1.00  ; 手动模式
OUT TR0
LD 703.04  ; #3腔体氦检阀开[SW]
OR D1148.12  ; #3腔体机构开始#3-1氦检（标漏步）
OR D1149.04  ; #3腔体机构开始#3-2氦检（标漏步）
ANDLD
DIFU(013) 303.04  ; #3腔体氦检阀开[Pls]
LD TR0
LD 303.04  ; #3腔体氦检阀开[Pls]
OR 403.04  ; #3腔体氦检阀开[M]
ANDLD
ANDNOT 313.04  ; #3腔体氦检阀关[Pls]
ANDNOT 803.04  ; #3腔体氦检阀开到位标志[0003.04]
AND D1122.14  ; #3腔体氦检阀打开允许条件
OUT 403.04  ; #3腔体氦检阀开[M]
LD TR0
LD 713.04  ; #3腔体氦检阀关[SW]
OR D1137.01  ; #3腔体关闭除破真空阀以外全部阀门（复位）
OR D1148.13  ; #3腔体机构关#3腔体氦检阀（标漏步）
OR D1149.05  ; #3腔体机构关#3腔体氦检阀（标漏步）
ANDLD
DIFU(013) 313.04  ; #3腔体氦检阀关[Pls]
LD TR0
LD 313.04  ; #3腔体氦检阀关[Pls]
OR 413.04  ; #3腔体氦检阀关[M]
ANDLD
ANDNOT 303.04  ; #3腔体氦检阀开[Pls]
ANDNOT 803.05  ; #3腔体氦检阀关到位标志[0003.05]
OUT 413.04  ; #3腔体氦检阀关[M]

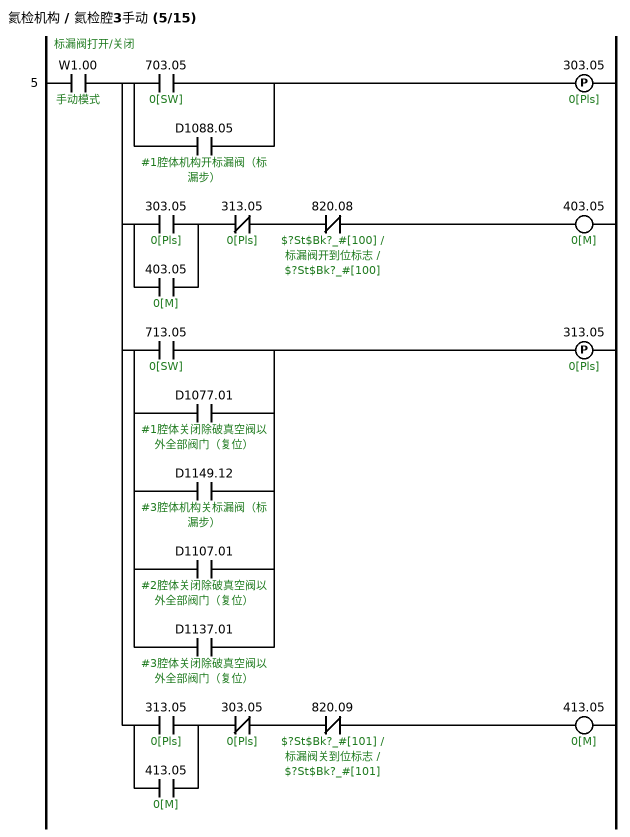
; rung 5: 标漏阀打开/关闭
LD W1.00  ; 手动模式
OUT TR0
LD 703.05  ; 0[SW]
OR D1088.05  ; #1腔体机构开标漏阀（标漏步）
ANDLD
DIFU(013) 303.05  ; 0[Pls]
LD TR0
LD 303.05  ; 0[Pls]
OR 403.05  ; 0[M]
ANDLD
ANDNOT 313.05  ; 0[Pls]
ANDNOT 820.08  ; $?St$Bk?_#[100] / 标漏阀开到位标志 / $?St$Bk?_#[100]
OUT 403.05  ; 0[M]
LD TR0
LD 713.05  ; 0[SW]
OR D1077.01  ; #1腔体关闭除破真空阀以外全部阀门（复位）
OR D1149.12  ; #3腔体机构关标漏阀（标漏步）
OR D1107.01  ; #2腔体关闭除破真空阀以外全部阀门（复位）
OR D1137.01  ; #3腔体关闭除破真空阀以外全部阀门（复位）
ANDLD
DIFU(013) 313.05  ; 0[Pls]
LD TR0
LD 313.05  ; 0[Pls]
OR 413.05  ; 0[M]
ANDLD
ANDNOT 303.05  ; 0[Pls]
ANDNOT 820.09  ; $?St$Bk?_#[101] / 标漏阀关到位标志 / $?St$Bk?_#[101]
OUT 413.05  ; 0[M]

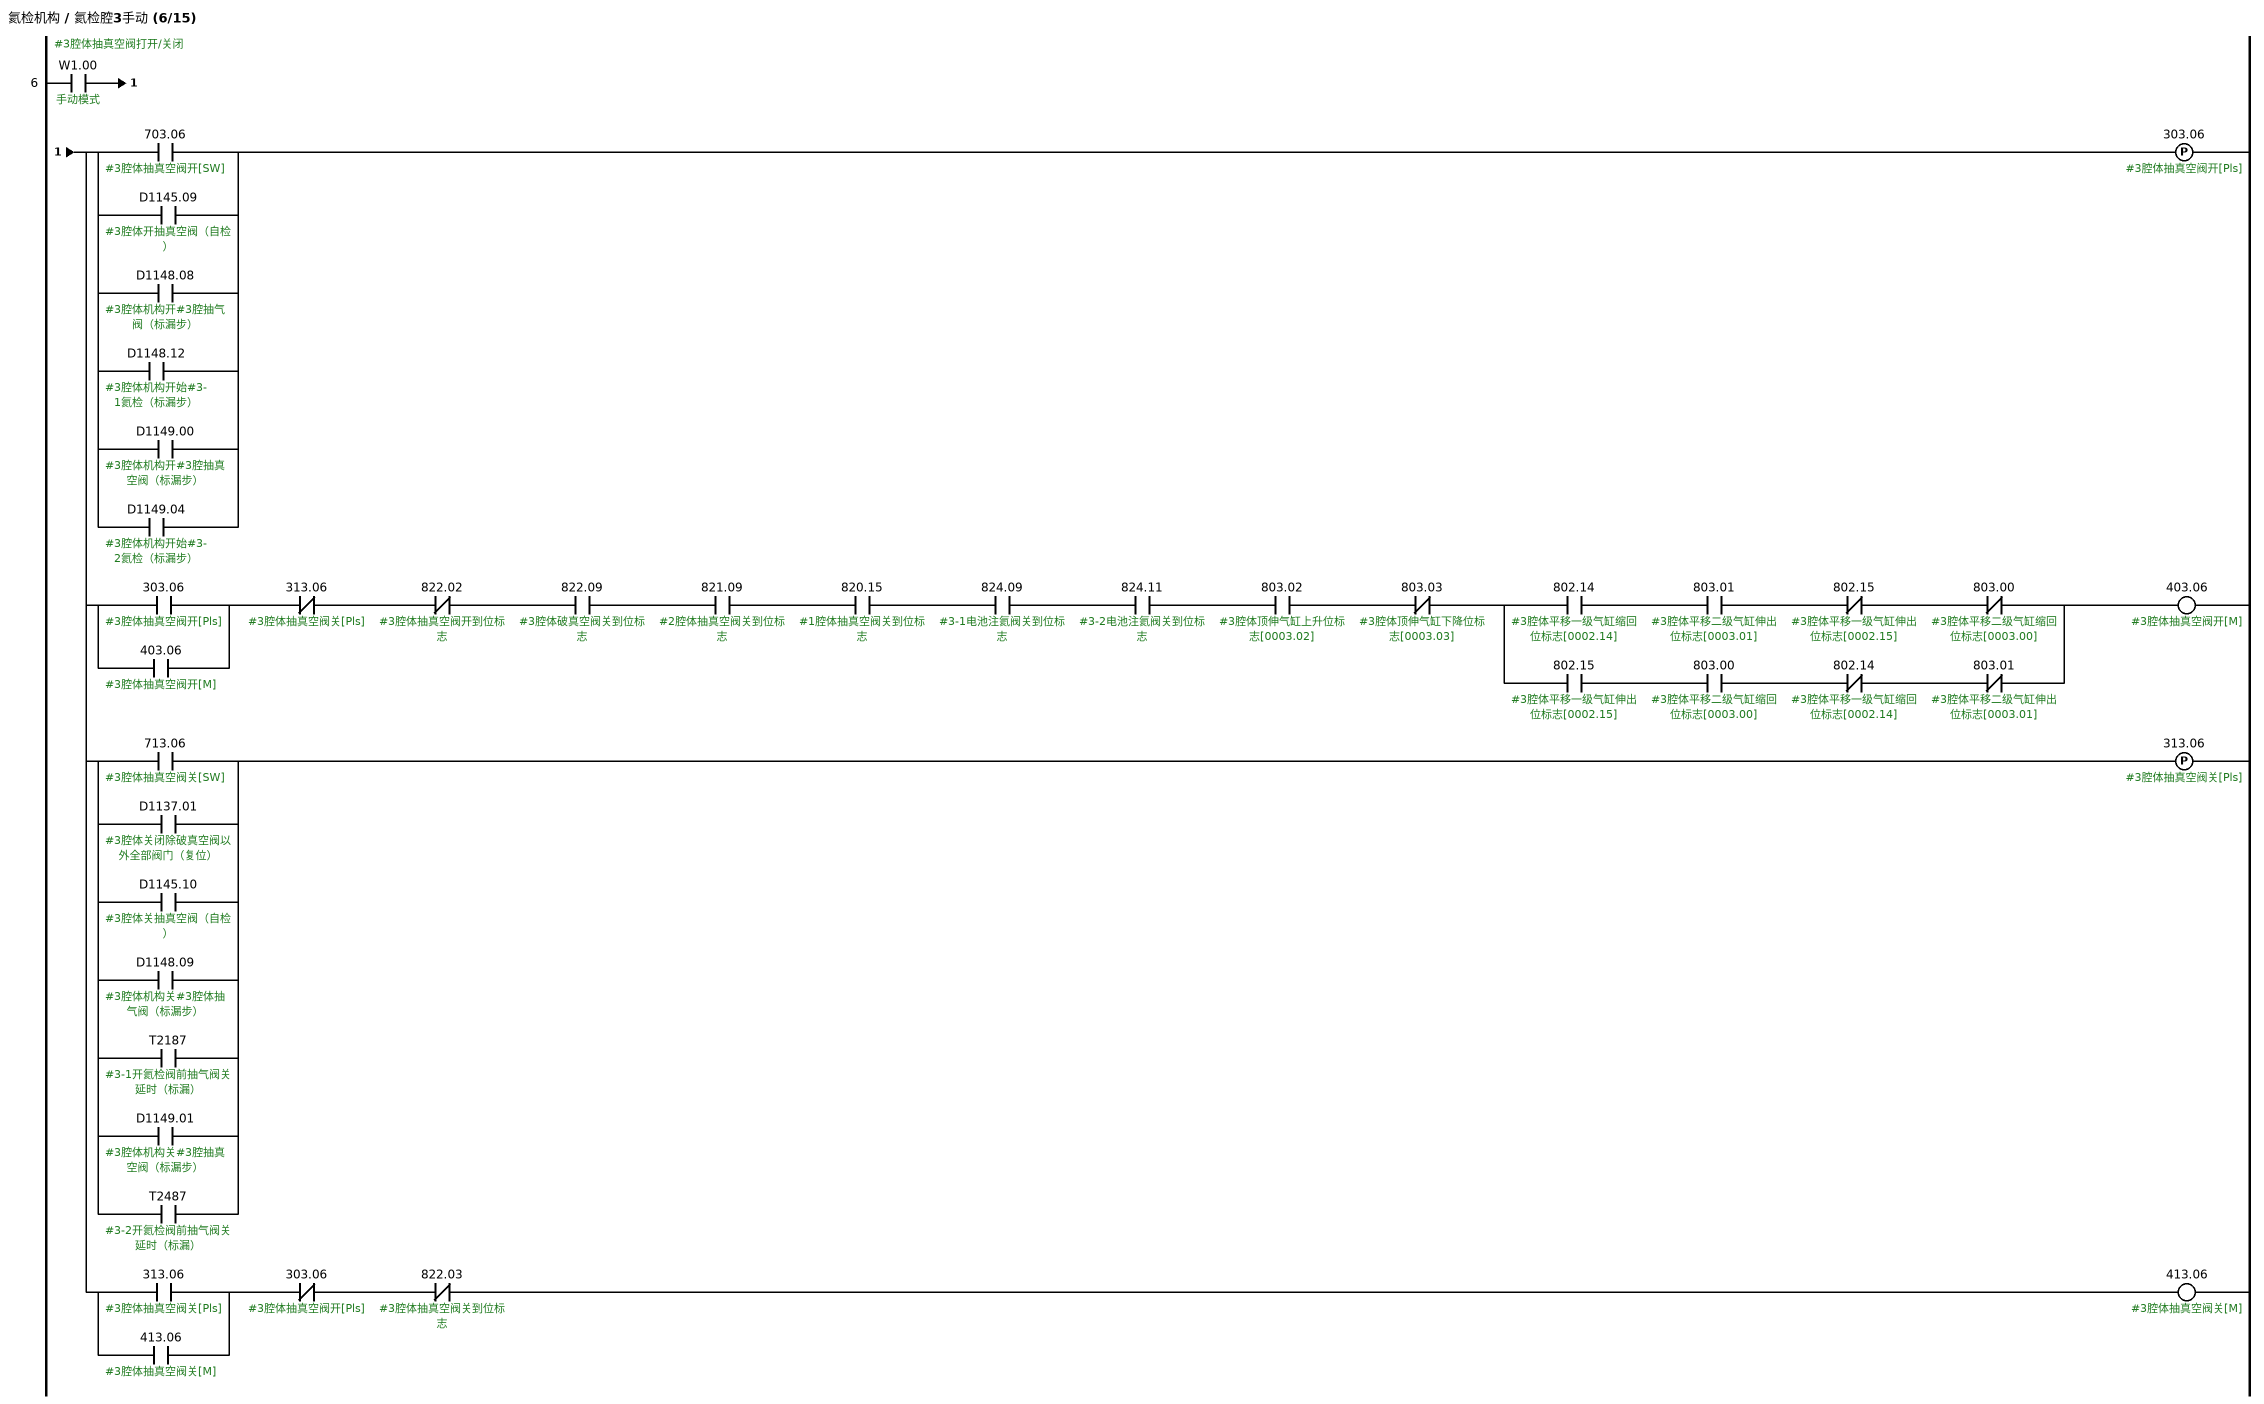
; rung 6: #3腔体抽真空阀打开/关闭
LD W1.00  ; 手动模式
OUT TR0
LD 703.06  ; #3腔体抽真空阀开[SW]
OR D1145.09  ; #3腔体开抽真空阀（自检）
OR D1148.08  ; #3腔体机构开#3腔抽气阀（标漏步）
OR D1148.12  ; #3腔体机构开始#3-1氦检（标漏步）
OR D1149.00  ; #3腔体机构开#3腔抽真空阀（标漏步）
OR D1149.04  ; #3腔体机构开始#3-2氦检（标漏步）
ANDLD
DIFU(013) 303.06  ; #3腔体抽真空阀开[Pls]
LD TR0
LD 303.06  ; #3腔体抽真空阀开[Pls]
OR 403.06  ; #3腔体抽真空阀开[M]
ANDLD
ANDNOT 313.06  ; #3腔体抽真空阀关[Pls]
ANDNOT 822.02  ; #3腔体抽真空阀开到位标志
AND 822.09  ; #3腔体破真空阀关到位标志
AND 821.09  ; #2腔体抽真空阀关到位标志
AND 820.15  ; #1腔体抽真空阀关到位标志
AND 824.09  ; #3-1电池注氦阀关到位标志
AND 824.11  ; #3-2电池注氦阀关到位标志
AND 803.02  ; #3腔体顶伸气缸上升位标志[0003.02]
ANDNOT 803.03  ; #3腔体顶伸气缸下降位标志[0003.03]
LD 802.14  ; #3腔体平移一级气缸缩回位标志[0002.14]
AND 803.01  ; #3腔体平移二级气缸伸出位标志[0003.01]
ANDNOT 802.15  ; #3腔体平移一级气缸伸出位标志[0002.15]
ANDNOT 803.00  ; #3腔体平移二级气缸缩回位标志[0003.00]
LD 802.15  ; #3腔体平移一级气缸伸出位标志[0002.15]
AND 803.00  ; #3腔体平移二级气缸缩回位标志[0003.00]
ANDNOT 802.14  ; #3腔体平移一级气缸缩回位标志[0002.14]
ANDNOT 803.01  ; #3腔体平移二级气缸伸出位标志[0003.01]
ORLD
ANDLD
OUT 403.06  ; #3腔体抽真空阀开[M]
LD TR0
LD 713.06  ; #3腔体抽真空阀关[SW]
OR D1137.01  ; #3腔体关闭除破真空阀以外全部阀门（复位）
OR D1145.10  ; #3腔体关抽真空阀（自检）
OR D1148.09  ; #3腔体机构关#3腔体抽气阀（标漏步）
OR T2187  ; #3-1开氦检阀前抽气阀关延时（标漏）
OR D1149.01  ; #3腔体机构关#3腔抽真空阀（标漏步）
OR T2487  ; #3-2开氦检阀前抽气阀关延时（标漏）
ANDLD
DIFU(013) 313.06  ; #3腔体抽真空阀关[Pls]
LD TR0
LD 313.06  ; #3腔体抽真空阀关[Pls]
OR 413.06  ; #3腔体抽真空阀关[M]
ANDLD
ANDNOT 303.06  ; #3腔体抽真空阀开[Pls]
ANDNOT 822.03  ; #3腔体抽真空阀关到位标志
OUT 413.06  ; #3腔体抽真空阀关[M]

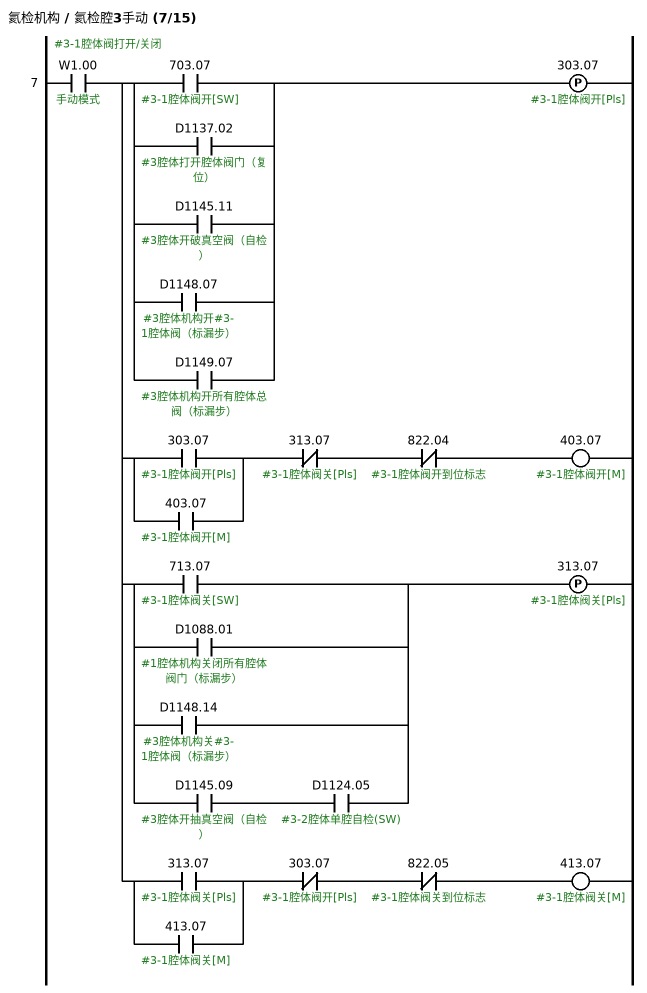
; rung 7: #3-1腔体阀打开/关闭
LD W1.00  ; 手动模式
OUT TR0
LD 703.07  ; #3-1腔体阀开[SW]
OR D1137.02  ; #3腔体打开腔体阀门（复位）
OR D1145.11  ; #3腔体开破真空阀（自检）
OR D1148.07  ; #3腔体机构开#3-1腔体阀（标漏步）
OR D1149.07  ; #3腔体机构开所有腔体总阀（标漏步）
ANDLD
DIFU(013) 303.07  ; #3-1腔体阀开[Pls]
LD TR0
LD 303.07  ; #3-1腔体阀开[Pls]
OR 403.07  ; #3-1腔体阀开[M]
ANDLD
ANDNOT 313.07  ; #3-1腔体阀关[Pls]
ANDNOT 822.04  ; #3-1腔体阀开到位标志
OUT 403.07  ; #3-1腔体阀开[M]
LD TR0
LD 713.07  ; #3-1腔体阀关[SW]
OR D1088.01  ; #1腔体机构关闭所有腔体阀门（标漏步）
OR D1148.14  ; #3腔体机构关#3-1腔体阀（标漏步）
LD D1145.09  ; #3腔体开抽真空阀（自检）
AND D1124.05  ; #3-2腔体单腔自检(SW)
ORLD
ANDLD
DIFU(013) 313.07  ; #3-1腔体阀关[Pls]
LD TR0
LD 313.07  ; #3-1腔体阀关[Pls]
OR 413.07  ; #3-1腔体阀关[M]
ANDLD
ANDNOT 303.07  ; #3-1腔体阀开[Pls]
ANDNOT 822.05  ; #3-1腔体阀关到位标志
OUT 413.07  ; #3-1腔体阀关[M]

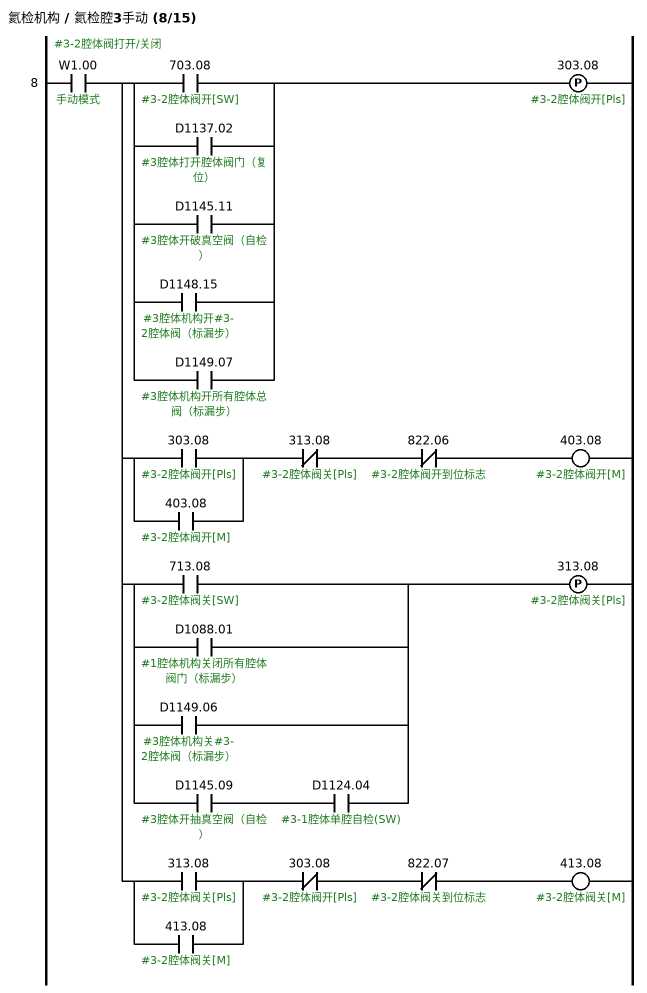
; rung 8: #3-2腔体阀打开/关闭
LD W1.00  ; 手动模式
OUT TR0
LD 703.08  ; #3-2腔体阀开[SW]
OR D1137.02  ; #3腔体打开腔体阀门（复位）
OR D1145.11  ; #3腔体开破真空阀（自检）
OR D1148.15  ; #3腔体机构开#3-2腔体阀（标漏步）
OR D1149.07  ; #3腔体机构开所有腔体总阀（标漏步）
ANDLD
DIFU(013) 303.08  ; #3-2腔体阀开[Pls]
LD TR0
LD 303.08  ; #3-2腔体阀开[Pls]
OR 403.08  ; #3-2腔体阀开[M]
ANDLD
ANDNOT 313.08  ; #3-2腔体阀关[Pls]
ANDNOT 822.06  ; #3-2腔体阀开到位标志
OUT 403.08  ; #3-2腔体阀开[M]
LD TR0
LD 713.08  ; #3-2腔体阀关[SW]
OR D1088.01  ; #1腔体机构关闭所有腔体阀门（标漏步）
OR D1149.06  ; #3腔体机构关#3-2腔体阀（标漏步）
LD D1145.09  ; #3腔体开抽真空阀（自检）
AND D1124.04  ; #3-1腔体单腔自检(SW)
ORLD
ANDLD
DIFU(013) 313.08  ; #3-2腔体阀关[Pls]
LD TR0
LD 313.08  ; #3-2腔体阀关[Pls]
OR 413.08  ; #3-2腔体阀关[M]
ANDLD
ANDNOT 303.08  ; #3-2腔体阀开[Pls]
ANDNOT 822.07  ; #3-2腔体阀关到位标志
OUT 413.08  ; #3-2腔体阀关[M]

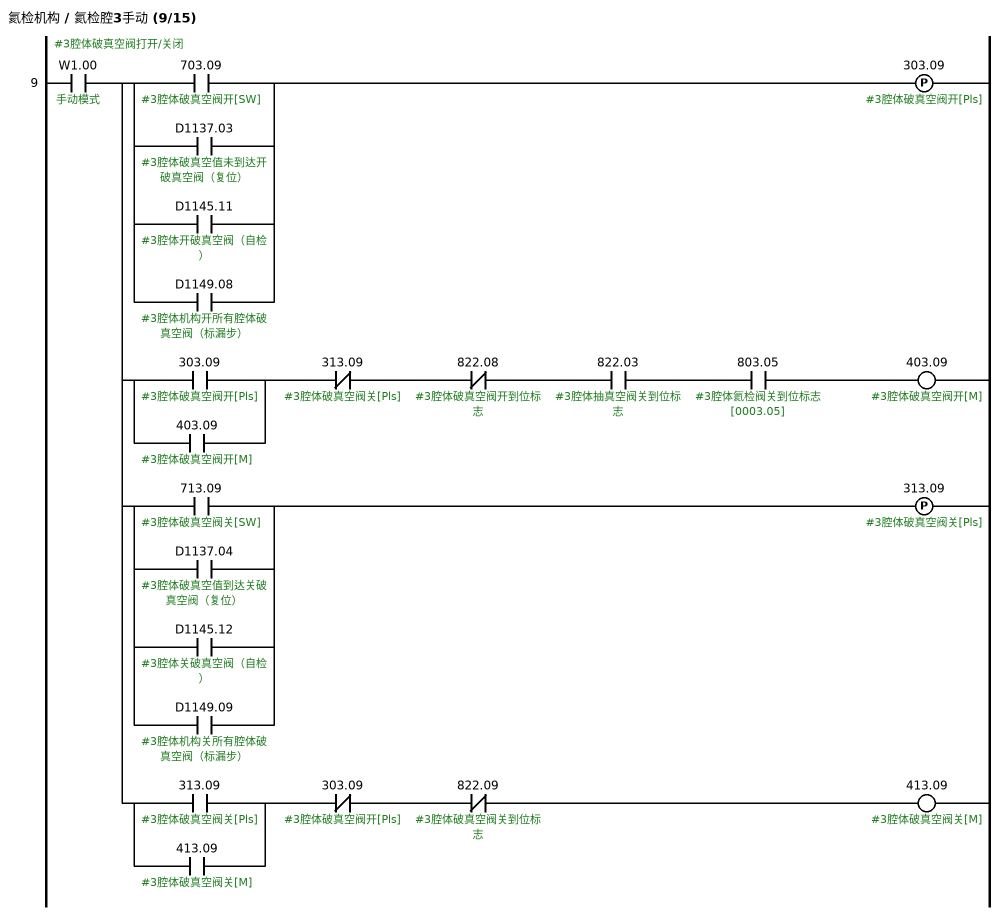
; rung 9: #3腔体破真空阀打开/关闭
LD W1.00  ; 手动模式
OUT TR0
LD 703.09  ; #3腔体破真空阀开[SW]
OR D1137.03  ; #3腔体破真空值未到达开破真空阀（复位）
OR D1145.11  ; #3腔体开破真空阀（自检）
OR D1149.08  ; #3腔体机构开所有腔体破真空阀（标漏步）
ANDLD
DIFU(013) 303.09  ; #3腔体破真空阀开[Pls]
LD TR0
LD 303.09  ; #3腔体破真空阀开[Pls]
OR 403.09  ; #3腔体破真空阀开[M]
ANDLD
ANDNOT 313.09  ; #3腔体破真空阀关[Pls]
ANDNOT 822.08  ; #3腔体破真空阀开到位标志
AND 822.03  ; #3腔体抽真空阀关到位标志
AND 803.05  ; #3腔体氦检阀关到位标志[0003.05]
OUT 403.09  ; #3腔体破真空阀开[M]
LD TR0
LD 713.09  ; #3腔体破真空阀关[SW]
OR D1137.04  ; #3腔体破真空值到达关破真空阀（复位）
OR D1145.12  ; #3腔体关破真空阀（自检）
OR D1149.09  ; #3腔体机构关所有腔体破真空阀（标漏步）
ANDLD
DIFU(013) 313.09  ; #3腔体破真空阀关[Pls]
LD TR0
LD 313.09  ; #3腔体破真空阀关[Pls]
OR 413.09  ; #3腔体破真空阀关[M]
ANDLD
ANDNOT 303.09  ; #3腔体破真空阀开[Pls]
ANDNOT 822.09  ; #3腔体破真空阀关到位标志
OUT 413.09  ; #3腔体破真空阀关[M]

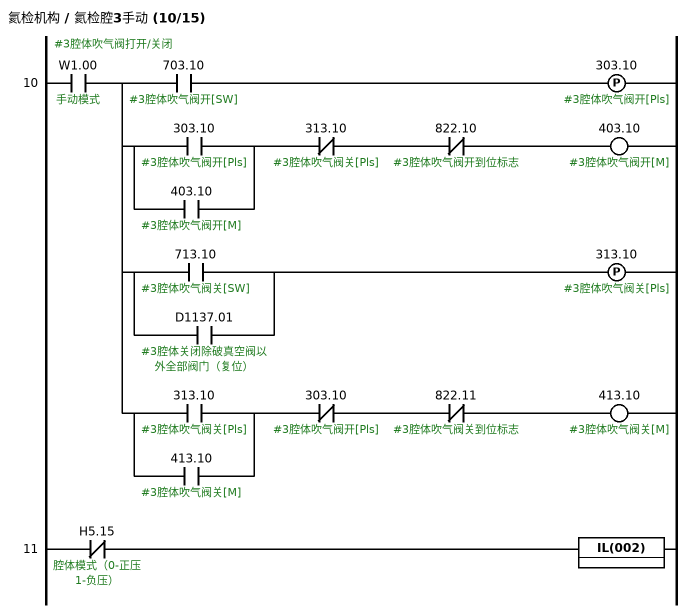
; rung 10: #3腔体吹气阀打开/关闭
LD W1.00  ; 手动模式
OUT TR0
AND 703.10  ; #3腔体吹气阀开[SW]
DIFU(013) 303.10  ; #3腔体吹气阀开[Pls]
LD TR0
LD 303.10  ; #3腔体吹气阀开[Pls]
OR 403.10  ; #3腔体吹气阀开[M]
ANDLD
ANDNOT 313.10  ; #3腔体吹气阀关[Pls]
ANDNOT 822.10  ; #3腔体吹气阀开到位标志
OUT 403.10  ; #3腔体吹气阀开[M]
LD TR0
LD 713.10  ; #3腔体吹气阀关[SW]
OR D1137.01  ; #3腔体关闭除破真空阀以外全部阀门（复位）
ANDLD
DIFU(013) 313.10  ; #3腔体吹气阀关[Pls]
LD TR0
LD 313.10  ; #3腔体吹气阀关[Pls]
OR 413.10  ; #3腔体吹气阀关[M]
ANDLD
ANDNOT 303.10  ; #3腔体吹气阀开[Pls]
ANDNOT 822.11  ; #3腔体吹气阀关到位标志
OUT 413.10  ; #3腔体吹气阀关[M]
; rung 11
LDNOT H5.15  ; 腔体模式（0-正压 1-负压）
IL(002)

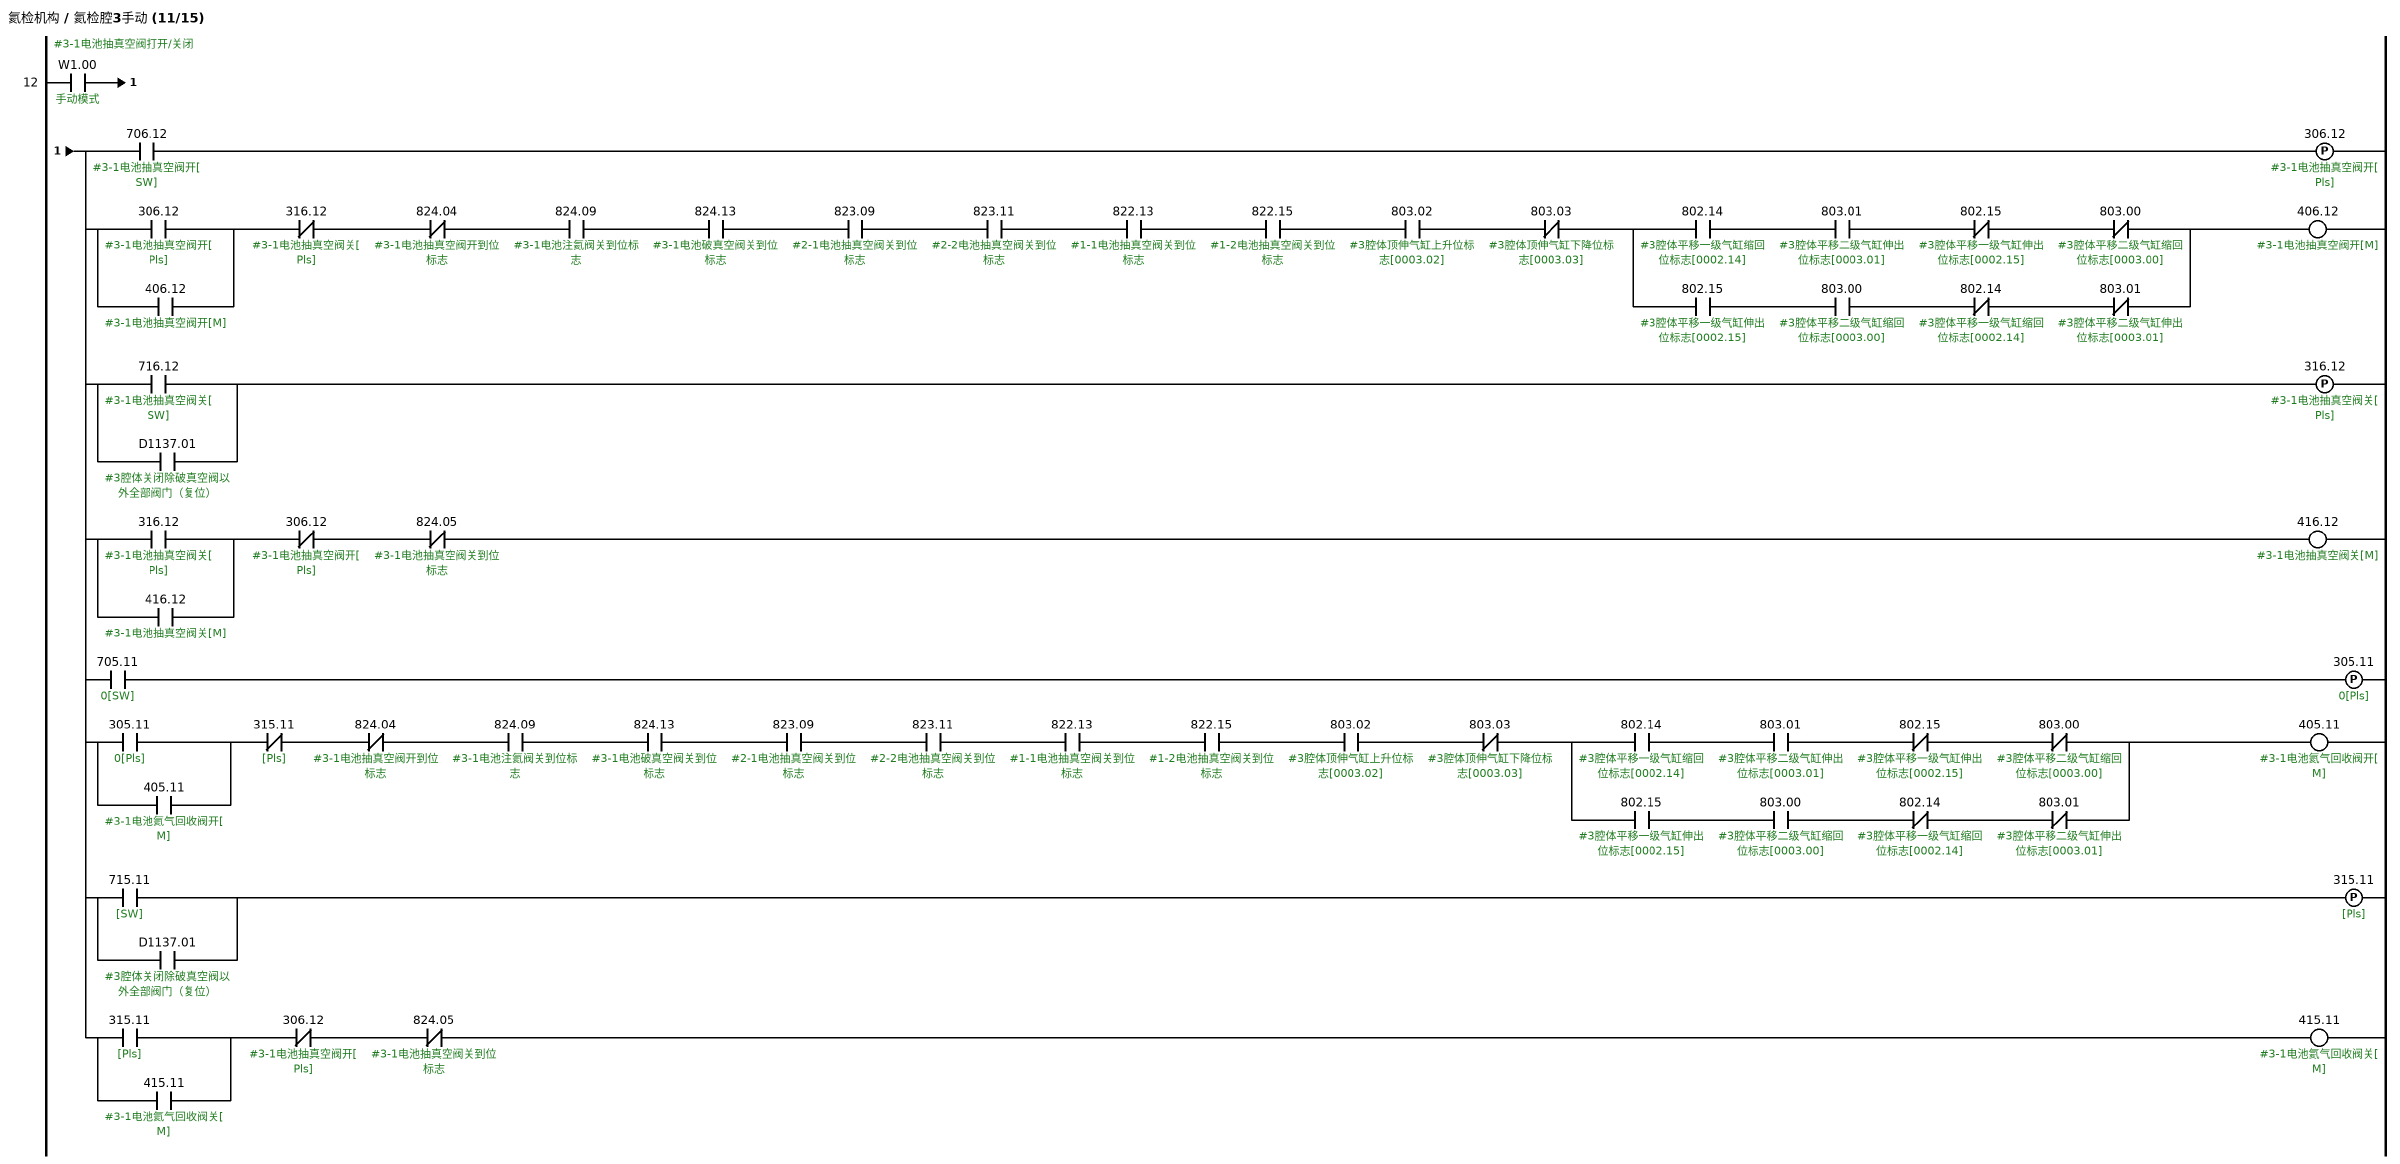
; rung 12: #3-1电池抽真空阀打开/关闭
LD W1.00  ; 手动模式
OUT TR0
AND 706.12  ; #3-1电池抽真空阀开[SW]
DIFU(013) 306.12  ; #3-1电池抽真空阀开[Pls]
LD TR0
LD 306.12  ; #3-1电池抽真空阀开[Pls]
OR 406.12  ; #3-1电池抽真空阀开[M]
ANDLD
ANDNOT 316.12  ; #3-1电池抽真空阀关[Pls]
ANDNOT 824.04  ; #3-1电池抽真空阀开到位标志
AND 824.09  ; #3-1电池注氦阀关到位标志
AND 824.13  ; #3-1电池破真空阀关到位标志
AND 823.09  ; #2-1电池抽真空阀关到位标志
AND 823.11  ; #2-2电池抽真空阀关到位标志
AND 822.13  ; #1-1电池抽真空阀关到位标志
AND 822.15  ; #1-2电池抽真空阀关到位标志
AND 803.02  ; #3腔体顶伸气缸上升位标志[0003.02]
ANDNOT 803.03  ; #3腔体顶伸气缸下降位标志[0003.03]
LD 802.14  ; #3腔体平移一级气缸缩回位标志[0002.14]
AND 803.01  ; #3腔体平移二级气缸伸出位标志[0003.01]
ANDNOT 802.15  ; #3腔体平移一级气缸伸出位标志[0002.15]
ANDNOT 803.00  ; #3腔体平移二级气缸缩回位标志[0003.00]
LD 802.15  ; #3腔体平移一级气缸伸出位标志[0002.15]
AND 803.00  ; #3腔体平移二级气缸缩回位标志[0003.00]
ANDNOT 802.14  ; #3腔体平移一级气缸缩回位标志[0002.14]
ANDNOT 803.01  ; #3腔体平移二级气缸伸出位标志[0003.01]
ORLD
ANDLD
OUT 406.12  ; #3-1电池抽真空阀开[M]
LD TR0
LD 716.12  ; #3-1电池抽真空阀关[SW]
OR D1137.01  ; #3腔体关闭除破真空阀以外全部阀门（复位）
ANDLD
DIFU(013) 316.12  ; #3-1电池抽真空阀关[Pls]
LD TR0
LD 316.12  ; #3-1电池抽真空阀关[Pls]
OR 416.12  ; #3-1电池抽真空阀关[M]
ANDLD
ANDNOT 306.12  ; #3-1电池抽真空阀开[Pls]
ANDNOT 824.05  ; #3-1电池抽真空阀关到位标志
OUT 416.12  ; #3-1电池抽真空阀关[M]
LD TR0
AND 705.11  ; 0[SW]
DIFU(013) 305.11  ; 0[Pls]
LD TR0
LD 305.11  ; 0[Pls]
OR 405.11  ; #3-1电池氦气回收阀开[M]
ANDLD
ANDNOT 315.11  ; [Pls]
ANDNOT 824.04  ; #3-1电池抽真空阀开到位标志
AND 824.09  ; #3-1电池注氦阀关到位标志
AND 824.13  ; #3-1电池破真空阀关到位标志
AND 823.09  ; #2-1电池抽真空阀关到位标志
AND 823.11  ; #2-2电池抽真空阀关到位标志
AND 822.13  ; #1-1电池抽真空阀关到位标志
AND 822.15  ; #1-2电池抽真空阀关到位标志
AND 803.02  ; #3腔体顶伸气缸上升位标志[0003.02]
ANDNOT 803.03  ; #3腔体顶伸气缸下降位标志[0003.03]
LD 802.14  ; #3腔体平移一级气缸缩回位标志[0002.14]
AND 803.01  ; #3腔体平移二级气缸伸出位标志[0003.01]
ANDNOT 802.15  ; #3腔体平移一级气缸伸出位标志[0002.15]
ANDNOT 803.00  ; #3腔体平移二级气缸缩回位标志[0003.00]
LD 802.15  ; #3腔体平移一级气缸伸出位标志[0002.15]
AND 803.00  ; #3腔体平移二级气缸缩回位标志[0003.00]
ANDNOT 802.14  ; #3腔体平移一级气缸缩回位标志[0002.14]
ANDNOT 803.01  ; #3腔体平移二级气缸伸出位标志[0003.01]
ORLD
ANDLD
OUT 405.11  ; #3-1电池氦气回收阀开[M]
LD TR0
LD 715.11  ; [SW]
OR D1137.01  ; #3腔体关闭除破真空阀以外全部阀门（复位）
ANDLD
DIFU(013) 315.11  ; [Pls]
LD TR0
LD 315.11  ; [Pls]
OR 415.11  ; #3-1电池氦气回收阀关[M]
ANDLD
ANDNOT 306.12  ; #3-1电池抽真空阀开[Pls]
ANDNOT 824.05  ; #3-1电池抽真空阀关到位标志
OUT 415.11  ; #3-1电池氦气回收阀关[M]

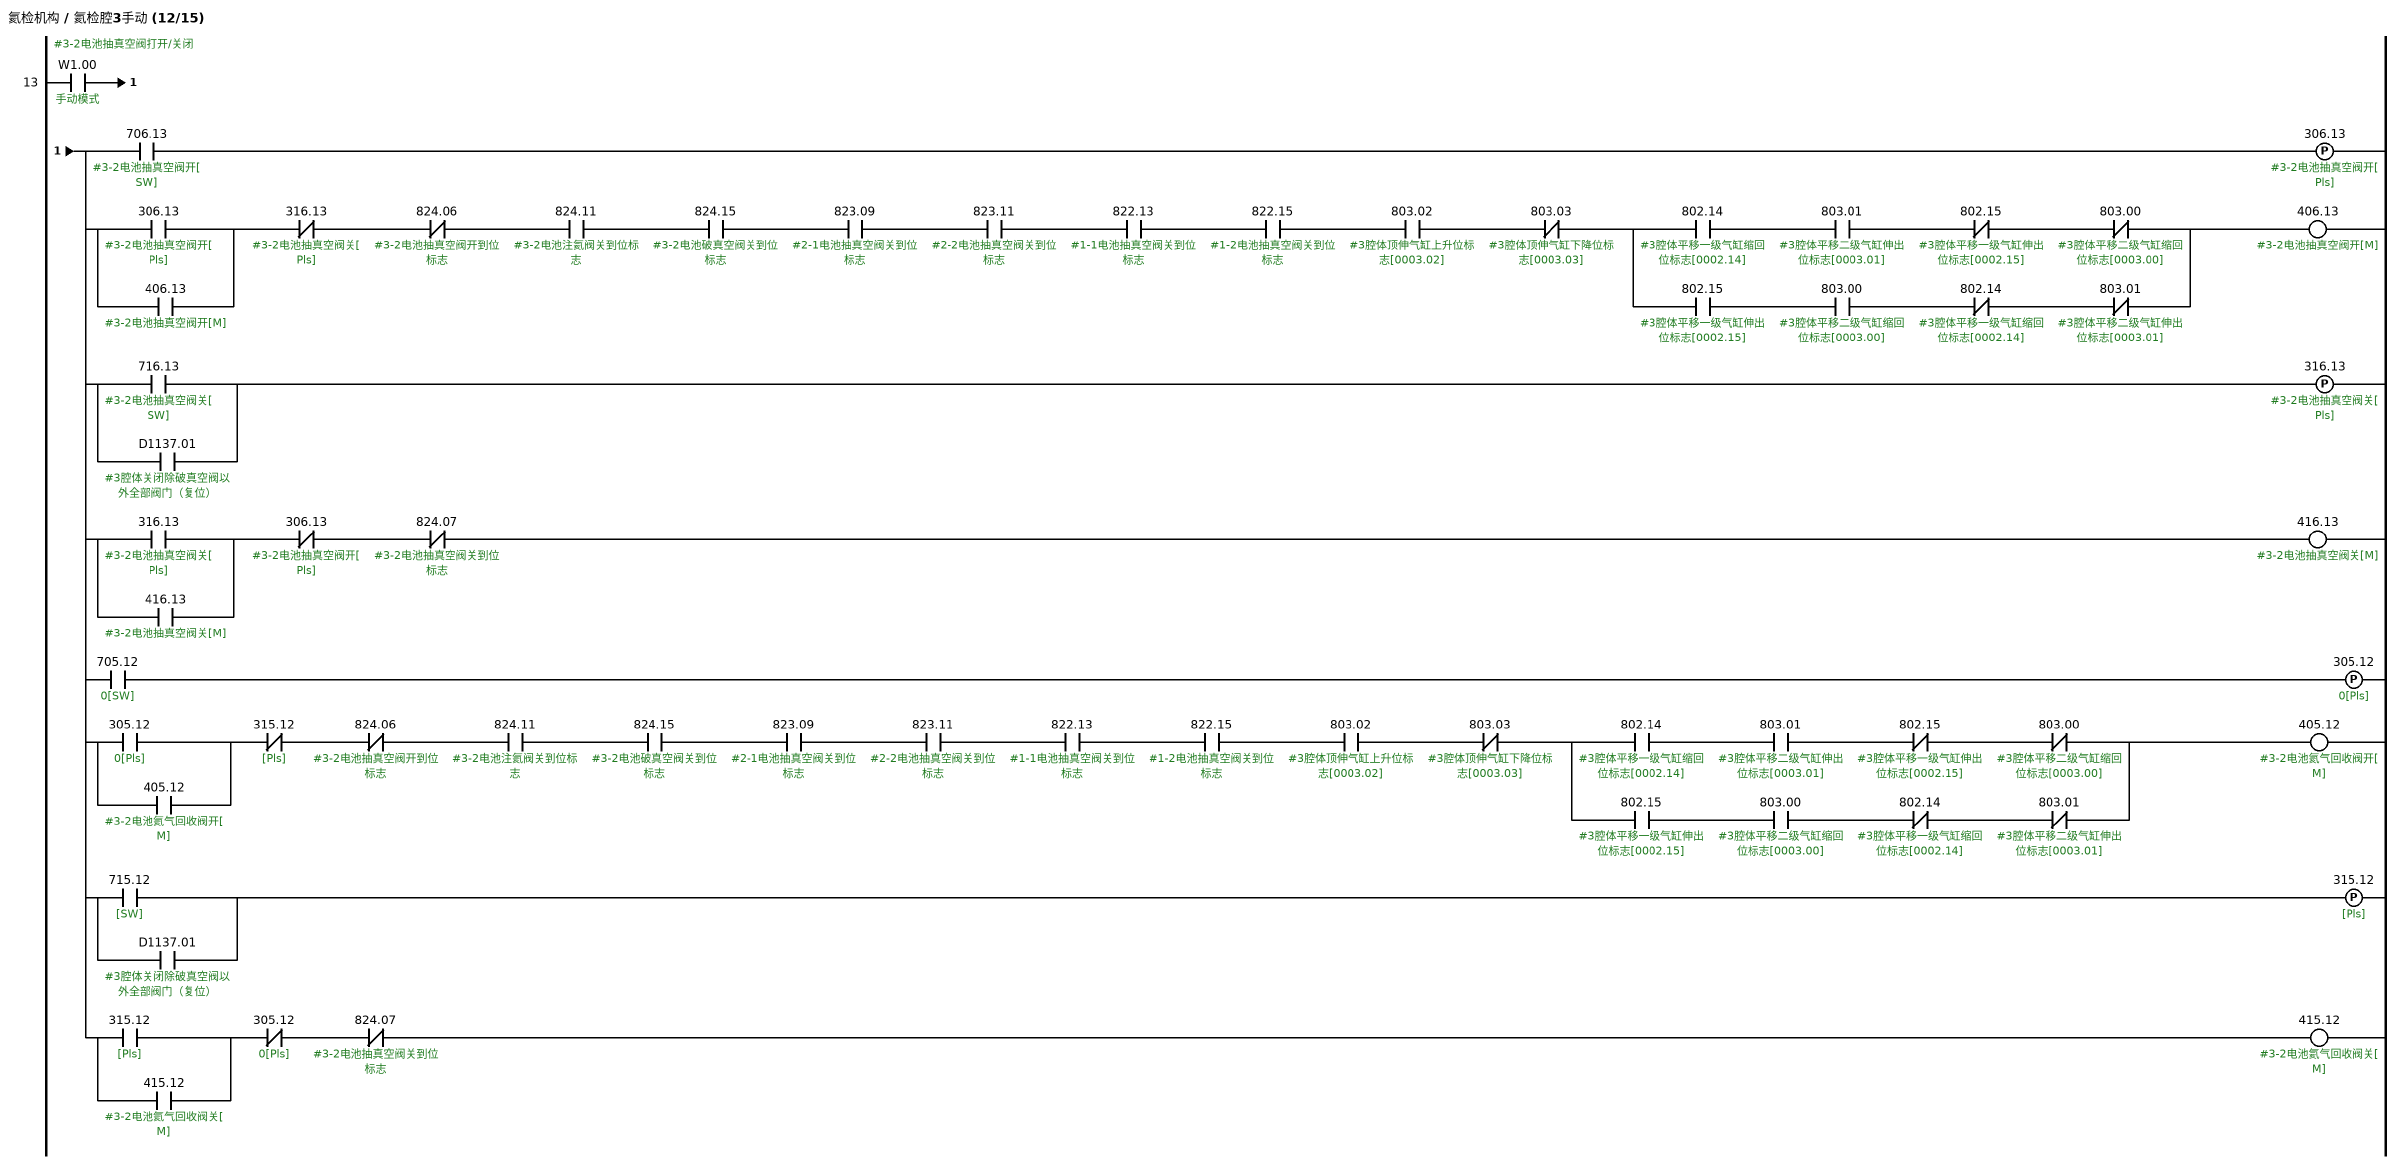
; rung 13: #3-2电池抽真空阀打开/关闭
LD W1.00  ; 手动模式
OUT TR0
AND 706.13  ; #3-2电池抽真空阀开[SW]
DIFU(013) 306.13  ; #3-2电池抽真空阀开[Pls]
LD TR0
LD 306.13  ; #3-2电池抽真空阀开[Pls]
OR 406.13  ; #3-2电池抽真空阀开[M]
ANDLD
ANDNOT 316.13  ; #3-2电池抽真空阀关[Pls]
ANDNOT 824.06  ; #3-2电池抽真空阀开到位标志
AND 824.11  ; #3-2电池注氦阀关到位标志
AND 824.15  ; #3-2电池破真空阀关到位标志
AND 823.09  ; #2-1电池抽真空阀关到位标志
AND 823.11  ; #2-2电池抽真空阀关到位标志
AND 822.13  ; #1-1电池抽真空阀关到位标志
AND 822.15  ; #1-2电池抽真空阀关到位标志
AND 803.02  ; #3腔体顶伸气缸上升位标志[0003.02]
ANDNOT 803.03  ; #3腔体顶伸气缸下降位标志[0003.03]
LD 802.14  ; #3腔体平移一级气缸缩回位标志[0002.14]
AND 803.01  ; #3腔体平移二级气缸伸出位标志[0003.01]
ANDNOT 802.15  ; #3腔体平移一级气缸伸出位标志[0002.15]
ANDNOT 803.00  ; #3腔体平移二级气缸缩回位标志[0003.00]
LD 802.15  ; #3腔体平移一级气缸伸出位标志[0002.15]
AND 803.00  ; #3腔体平移二级气缸缩回位标志[0003.00]
ANDNOT 802.14  ; #3腔体平移一级气缸缩回位标志[0002.14]
ANDNOT 803.01  ; #3腔体平移二级气缸伸出位标志[0003.01]
ORLD
ANDLD
OUT 406.13  ; #3-2电池抽真空阀开[M]
LD TR0
LD 716.13  ; #3-2电池抽真空阀关[SW]
OR D1137.01  ; #3腔体关闭除破真空阀以外全部阀门（复位）
ANDLD
DIFU(013) 316.13  ; #3-2电池抽真空阀关[Pls]
LD TR0
LD 316.13  ; #3-2电池抽真空阀关[Pls]
OR 416.13  ; #3-2电池抽真空阀关[M]
ANDLD
ANDNOT 306.13  ; #3-2电池抽真空阀开[Pls]
ANDNOT 824.07  ; #3-2电池抽真空阀关到位标志
OUT 416.13  ; #3-2电池抽真空阀关[M]
LD TR0
AND 705.12  ; 0[SW]
DIFU(013) 305.12  ; 0[Pls]
LD TR0
LD 305.12  ; 0[Pls]
OR 405.12  ; #3-2电池氦气回收阀开[M]
ANDLD
ANDNOT 315.12  ; [Pls]
ANDNOT 824.06  ; #3-2电池抽真空阀开到位标志
AND 824.11  ; #3-2电池注氦阀关到位标志
AND 824.15  ; #3-2电池破真空阀关到位标志
AND 823.09  ; #2-1电池抽真空阀关到位标志
AND 823.11  ; #2-2电池抽真空阀关到位标志
AND 822.13  ; #1-1电池抽真空阀关到位标志
AND 822.15  ; #1-2电池抽真空阀关到位标志
AND 803.02  ; #3腔体顶伸气缸上升位标志[0003.02]
ANDNOT 803.03  ; #3腔体顶伸气缸下降位标志[0003.03]
LD 802.14  ; #3腔体平移一级气缸缩回位标志[0002.14]
AND 803.01  ; #3腔体平移二级气缸伸出位标志[0003.01]
ANDNOT 802.15  ; #3腔体平移一级气缸伸出位标志[0002.15]
ANDNOT 803.00  ; #3腔体平移二级气缸缩回位标志[0003.00]
LD 802.15  ; #3腔体平移一级气缸伸出位标志[0002.15]
AND 803.00  ; #3腔体平移二级气缸缩回位标志[0003.00]
ANDNOT 802.14  ; #3腔体平移一级气缸缩回位标志[0002.14]
ANDNOT 803.01  ; #3腔体平移二级气缸伸出位标志[0003.01]
ORLD
ANDLD
OUT 405.12  ; #3-2电池氦气回收阀开[M]
LD TR0
LD 715.12  ; [SW]
OR D1137.01  ; #3腔体关闭除破真空阀以外全部阀门（复位）
ANDLD
DIFU(013) 315.12  ; [Pls]
LD TR0
LD 315.12  ; [Pls]
OR 415.12  ; #3-2电池氦气回收阀关[M]
ANDLD
ANDNOT 305.12  ; 0[Pls]
ANDNOT 824.07  ; #3-2电池抽真空阀关到位标志
OUT 415.12  ; #3-2电池氦气回收阀关[M]

